(* CODESYS project T620X_PLC_CR711S_SP16p5_32bit.project
   Title: T620X PLC
   Version: 1.0.3.0
   Company: Mtech

Project tree, tasks and I/O mapping:
  SafetyPLC : CR711S SIL2, ifm electronic, order no. CR711S, version 3.2.0.0
    application Application
      libraries: ifmR360-3, * (ifm electronic); Standard, * (System); Util, * (System)
      task Task (cyclic, interval t#10ms, priority 1, watchdog t#8ms x 1) calls PLC_PRG
      global variables EVL
      program PLC_PRG [FBD]
    Communication : Communication, ifm electronic, version 3.2.0.0
      CAN : CAN, ifm electronic, version 3.2.0.0
      Ethernet : Ethernet, ifm electronic, version 3.2.0.0
    HMI : HMI, ifm electronic, version 3.2.0.0
      User_LEDs : User_LEDs, ifm electronic, version 3.2.0.0
          input  UserLED0_I AT %IB534 : LED_IEC_B_INPUT_MAPPING_TYPE  // UserLED0_I
          input  UserLED1_I : LED_IEC_B_INPUT_MAPPING_TYPE  // UserLED1_I
          input  UserLED2_I : LED_IEC_B_INPUT_MAPPING_TYPE  // UserLED2_I
          input  UserLED3_I : LED_IEC_B_INPUT_MAPPING_TYPE  // UserLED3_I
          output UserLED0_Q : LED_IEC_B_OUTPUT_MAPPING_TYPE  // User LED 0
          output UserLED1_Q : LED_IEC_B_OUTPUT_MAPPING_TYPE  // User LED 1
          output UserLED2_Q : LED_IEC_B_OUTPUT_MAPPING_TYPE  // User LED 2
          output UserLED3_Q : LED_IEC_B_OUTPUT_MAPPING_TYPE  // User LED 3
    Local_IO : Local_IO, ifm electronic, version 3.2.0.0
      Inputs : Inputs, ifm electronic, version 3.2.0.0
          input  IN0100_I : IN_MULTIFUNCTION_A_INPUT_MAPPING_TYPE  // IN0100_I
          input  IN0101_I : IN_MULTIFUNCTION_A_INPUT_MAPPING_TYPE  // IN0101_I
          input  IN0102_I : IN_MULTIFUNCTION_A_INPUT_MAPPING_TYPE  // IN0102_I
          input  IN0103_I : IN_MULTIFUNCTION_A_INPUT_MAPPING_TYPE  // IN0103_I
          input  IN0200_I : IN_MULTIFUNCTION_A_INPUT_MAPPING_TYPE  // IN0200_I
          input  IN0201_I : IN_MULTIFUNCTION_A_INPUT_MAPPING_TYPE  // IN0201_I
          input  IN0202_I : IN_MULTIFUNCTION_A_INPUT_MAPPING_TYPE  // IN0202_I
          input  IN0203_I : IN_MULTIFUNCTION_A_INPUT_MAPPING_TYPE  // IN0203_I
          input  IN0600_I : IN_MULTIFUNCTION_A_INPUT_MAPPING_TYPE  // IN0600_I
          input  IN0601_I : IN_MULTIFUNCTION_A_INPUT_MAPPING_TYPE  // IN0601_I
          input  IN0602_I : IN_MULTIFUNCTION_A_INPUT_MAPPING_TYPE  // IN0602_I
          input  IN0603_I : IN_MULTIFUNCTION_A_INPUT_MAPPING_TYPE  // IN0603_I
          input  IN0700_I : IN_MULTIFUNCTION_A_INPUT_MAPPING_TYPE  // IN0700_I
          input  IN0701_I : IN_MULTIFUNCTION_A_INPUT_MAPPING_TYPE  // IN0701_I
          input  IN0702_I : IN_MULTIFUNCTION_A_INPUT_MAPPING_TYPE  // IN0702_I
          input  IN0703_I : IN_MULTIFUNCTION_A_INPUT_MAPPING_TYPE  // IN0703_I
          input  IN0400_I : IN_RESISTOR_A_INPUT_MAPPING_TYPE  // IN0400_I
          input  IN0401_I : IN_RESISTOR_A_INPUT_MAPPING_TYPE  // IN0401_I
          input  IN0900_I : IN_RESISTOR_A_INPUT_MAPPING_TYPE  // IN0900_I
          input  IN0901_I : IN_RESISTOR_A_INPUT_MAPPING_TYPE  // IN0901_I
          input  IN0300_I : IN_DIGITAL_B_INPUT_MAPPING_TYPE  // IN0300_I
          input  IN0301_I : IN_DIGITAL_B_INPUT_MAPPING_TYPE  // IN0301_I
          input  IN0800_I : IN_DIGITAL_B_INPUT_MAPPING_TYPE  // IN0800_I
          input  IN0801_I : IN_DIGITAL_B_INPUT_MAPPING_TYPE  // IN0801_I
          input  COM_RESET_I : IN_COMMUNICATION_RESET_INPUT_MAPPING_TYPE  // COM_RESET_I
          input  IN0000_I : IN_FREQUENCY_B_CHANNEL_A_INPUT_MAPPING_TYPE  // IN0000_I
          input  IN0002_I : IN_FREQUENCY_B_CHANNEL_A_INPUT_MAPPING_TYPE  // IN0002_I
          input  IN0500_I : IN_FREQUENCY_B_CHANNEL_A_INPUT_MAPPING_TYPE  // IN0500_I
          input  IN0502_I : IN_FREQUENCY_B_CHANNEL_A_INPUT_MAPPING_TYPE  // IN0502_I
          input  IN0001_I : IN_FREQUENCY_B_CHANNEL_B_INPUT_MAPPING_TYPE  // IN0001_I
          input  IN0003_I : IN_FREQUENCY_B_CHANNEL_B_INPUT_MAPPING_TYPE  // IN0003_I
          input  IN0501_I : IN_FREQUENCY_B_CHANNEL_B_INPUT_MAPPING_TYPE  // IN0501_I
          input  IN0503_I : IN_FREQUENCY_B_CHANNEL_B_INPUT_MAPPING_TYPE  // IN0503_I
      Outputs : Outputs, ifm electronic, version 3.2.0.0
          input  OUT0006_I : OUT_PWM_40_BRIDGE_A_INPUT_MAPPING_TYPE  // OUT0006_I
          input  OUT0106_I : OUT_PWM_40_BRIDGE_A_INPUT_MAPPING_TYPE  // OUT0106_I
          input  OUT0206_I : OUT_PWM_40_BRIDGE_A_INPUT_MAPPING_TYPE  // OUT0206_I
          input  OUT0008_I : OUT_PWM_40_A_INPUT_MAPPING_TYPE  // OUT0008_I
          input  OUT0108_I : OUT_PWM_40_A_INPUT_MAPPING_TYPE  // OUT0108_I
          input  OUT0208_I : OUT_PWM_40_A_INPUT_MAPPING_TYPE  // OUT0208_I
          input  OUT0000_I : OUT_PWM_25_A_INPUT_MAPPING_TYPE  // OUT0000_I
          input  OUT0002_I : OUT_PWM_25_A_INPUT_MAPPING_TYPE  // OUT0002_I
          input  OUT0004_I : OUT_PWM_25_A_INPUT_MAPPING_TYPE  // OUT0004_I
          input  OUT0100_I : OUT_PWM_25_A_INPUT_MAPPING_TYPE  // OUT0100_I
          input  OUT0102_I : OUT_PWM_25_A_INPUT_MAPPING_TYPE  // OUT0102_I
          input  OUT0104_I : OUT_PWM_25_A_INPUT_MAPPING_TYPE  // OUT0104_I
          input  OUT0200_I : OUT_PWM_25_A_INPUT_MAPPING_TYPE  // OUT0200_I
          input  OUT0202_I : OUT_PWM_25_A_INPUT_MAPPING_TYPE  // OUT0202_I
          input  OUT0204_I : OUT_PWM_25_A_INPUT_MAPPING_TYPE  // OUT0204_I
          input  OUT3001_I : OUT_VOLTAGE_A_INPUT_MAPPING_TYPE  // OUT3001_I
          input  OUT3000_I : OUT_SUPPLY_A_INPUT_MAPPING_TYPE  // OUT3000_I
          input  OUT0001_I : OUT_PWM_25_B_INPUT_MAPPING_TYPE  // OUT0001_I
          input  OUT0003_I : OUT_PWM_25_B_INPUT_MAPPING_TYPE  // OUT0003_I
          input  OUT0005_I : OUT_PWM_25_B_INPUT_MAPPING_TYPE  // OUT0005_I
          input  OUT0101_I : OUT_PWM_25_B_INPUT_MAPPING_TYPE  // OUT0101_I
          input  OUT0103_I : OUT_PWM_25_B_INPUT_MAPPING_TYPE  // OUT0103_I
          input  OUT0105_I : OUT_PWM_25_B_INPUT_MAPPING_TYPE  // OUT0105_I
          input  OUT0201_I : OUT_PWM_25_B_INPUT_MAPPING_TYPE  // OUT0201_I
          input  OUT0203_I : OUT_PWM_25_B_INPUT_MAPPING_TYPE  // OUT0203_I
          input  OUT0205_I : OUT_PWM_25_B_INPUT_MAPPING_TYPE  // OUT0205_I
          input  OUT0007_I : OUT_PWM_40_BRIDGE_A_INPUT_MAPPING_TYPE  // OUT0007_I
          input  OUT0107_I : OUT_PWM_40_BRIDGE_A_INPUT_MAPPING_TYPE  // OUT0107_I
          input  OUT0207_I : OUT_PWM_40_BRIDGE_A_INPUT_MAPPING_TYPE  // OUT0207_I
          output OUT0006_Q : OUT_PWM_40_BRIDGE_A_OUTPUT_MAPPING_TYPE  // OUT0006_Q
          output OUT0106_Q : OUT_PWM_40_BRIDGE_A_OUTPUT_MAPPING_TYPE  // OUT0106_Q
          output OUT0206_Q : OUT_PWM_40_BRIDGE_A_OUTPUT_MAPPING_TYPE  // OUT0206_Q
          output OUT0008_Q : OUT_PWM_40_A_OUTPUT_MAPPING_TYPE  // OUT0008_Q
          output OUT0108_Q : OUT_PWM_40_A_OUTPUT_MAPPING_TYPE  // OUT0108_Q
          output OUT0208_Q : OUT_PWM_40_A_OUTPUT_MAPPING_TYPE  // OUT0208_Q
          output OUT0000_Q : OUT_PWM_25_A_OUTPUT_MAPPING_TYPE  // OUT0000_Q
          output OUT0002_Q : OUT_PWM_25_A_OUTPUT_MAPPING_TYPE  // OUT0002_Q
          output OUT0004_Q : OUT_PWM_25_A_OUTPUT_MAPPING_TYPE  // OUT0004_Q
          output OUT0100_Q : OUT_PWM_25_A_OUTPUT_MAPPING_TYPE  // OUT0100_Q
          output OUT0102_Q : OUT_PWM_25_A_OUTPUT_MAPPING_TYPE  // OUT0102_Q
          output OUT0104_Q : OUT_PWM_25_A_OUTPUT_MAPPING_TYPE  // OUT0104_Q
          output OUT0200_Q : OUT_PWM_25_A_OUTPUT_MAPPING_TYPE  // OUT0200_Q
          output OUT0202_Q : OUT_PWM_25_A_OUTPUT_MAPPING_TYPE  // OUT0202_Q
          output OUT0204_Q : OUT_PWM_25_A_OUTPUT_MAPPING_TYPE  // OUT0204_Q
          output OUT3001_Q : OUT_VOLTAGE_A_OUTPUT_MAPPING_TYPE  // OUT3001_Q
          output OUT3000_Q : OUT_SUPPLY_A_OUTPUT_MAPPING_TYPE  // OUT3000_Q
          output OUT0001_Q : OUT_PWM_25_B_OUTPUT_MAPPING_TYPE  // OUT0001_Q
          output OUT0003_Q : OUT_PWM_25_B_OUTPUT_MAPPING_TYPE  // OUT0003_Q
          output OUT0005_Q : OUT_PWM_25_B_OUTPUT_MAPPING_TYPE  // OUT0005_Q
          output OUT0101_Q : OUT_PWM_25_B_OUTPUT_MAPPING_TYPE  // OUT0101_Q
          output OUT0103_Q : OUT_PWM_25_B_OUTPUT_MAPPING_TYPE  // OUT0103_Q
          output OUT0105_Q : OUT_PWM_25_B_OUTPUT_MAPPING_TYPE  // OUT0105_Q
          output OUT0201_Q : OUT_PWM_25_B_OUTPUT_MAPPING_TYPE  // OUT0201_Q
          output OUT0203_Q : OUT_PWM_25_B_OUTPUT_MAPPING_TYPE  // OUT0203_Q
          output OUT0205_Q : OUT_PWM_25_B_OUTPUT_MAPPING_TYPE  // OUT0205_Q
          output OUT0007_Q : OUT_PWM_40_BRIDGE_A_OUTPUT_MAPPING_TYPE  // OUT0007_Q
          output OUT0107_Q : OUT_PWM_40_BRIDGE_A_OUTPUT_MAPPING_TYPE  // OUT0107_Q
          output OUT0207_Q : OUT_PWM_40_BRIDGE_A_OUTPUT_MAPPING_TYPE  // OUT0207_Q
      System_Inputs : System_Inputs, ifm electronic, version 3.2.0.0
          input  VBB30 : IN_SYSTEM_VOLTAGE_INPUT_MAPPING_TYPE  // VBB30
          input  VBB15 : IN_SYSTEM_VOLTAGE_INPUT_MAPPING_TYPE  // VBB15
          input  TemperatureBoard0 : IN_TEMPERATURE_INPUT_MAPPING_TYPE  // TemperatureBoard0
          input  TemperatureChip0 : IN_TEMPERATURE_INPUT_MAPPING_TYPE  // TemperatureChip0
      System_Outputs : System_Outputs, ifm electronic, version 3.2.0.0
          input  VBB0_SW_I : OUT_GROUP_SWITCH_INPUT_MAPPING_TYPE  // VBB0_SW_I
          input  VBB1_SW_I : OUT_GROUP_SWITCH_INPUT_MAPPING_TYPE  // VBB1_SW_I
          input  VBB2_SW_I : OUT_GROUP_SWITCH_INPUT_MAPPING_TYPE  // VBB2_SW_I
          output VBB0_SW_Q : OUT_GROUP_SWITCH_OUTPUT_MAPPING_TYPE  // VBB0_SW_Q
          output VBB1_SW_Q : OUT_GROUP_SWITCH_OUTPUT_MAPPING_TYPE  // VBB1_SW_Q
          output VBB2_SW_Q : OUT_GROUP_SWITCH_OUTPUT_MAPPING_TYPE  // VBB2_SW_Q
          output SUPPLY_SWITCH_Q : OUT_SYS_SWITCH_OUTPUT_MAPPING_TYPE  // SUPPLY_SWITCH_Q
  StandardPLC : CR711S Standard, ifm electronic, order no. CR711S, version 3.2.0.0
    application Application
      libraries: ifmR360-3, * (ifm electronic); Standard, * (System); Util, * (System); PIL Master Library, 1.0.0 (Powerhouse IRL Ltd); SLL_IFM_Version, 0.0.0.2 (SLL); SLL_IFM_CRXXXX, 0.0.0.1 (SLL); SLL Common, 0.0.0.1 (SLL); SLL_IFM_IO, 0.0.1.0 (SLL)
      task Task (cyclic, interval t#10ms, priority 1, watchdog t#8ms x 1) calls PLC_PRG_MAIN
      task Task_UDP (cyclic, interval 2 ms, priority 2, watchdog T#500MS x 1) calls UDP_MAIN
      EVC
      program PLC_Version [FBD]
      global variables NVL_UDP_TX
      Inputs/
        program Inputs [FBD]
      program UDP_MAIN [FBD]
      declarations NVL_UDP_RX
      Outputs/
        program Outputs [FBD]
        function block CRXXXX_OUTPUT_PWM_FB [FBD]: Process
      Visualisations/
        visualisation Input_IFM_PLC_CRXXXX
        visualisation Output_IFM_PLC_CRXXXX
        visualisation Output_IFM_PLC_CRXXXX_GROUP
        visualisation Inputs_Test
        visualisation Outputs_Test
      program PLC_UDP_WDT_Check [FBD]
      data type T620X_SETTINGS
      App_PLC/
        program PLC_PRG_MAIN [FBD]
        global variables GVL_APP
        Control/
          program TRACK [FBD]
          program INTERLOCKS [FBD]
        program PLC_PRG_APP [FBD]
    Communication : Communication, ifm electronic, version 3.2.0.0
      CAN : CAN, ifm electronic, version 3.2.0.0
      Ethernet : Ethernet, ifm electronic, version 3.2.0.0
    HMI : HMI, ifm electronic, version 3.2.0.0
      User_LEDs : User_LEDs, ifm electronic, version 3.2.0.0
          input  UserLED0_I : LED_IEC_B_INPUT_MAPPING_TYPE  // UserLED0_I
          input  UserLED1_I : LED_IEC_B_INPUT_MAPPING_TYPE  // UserLED1_I
          input  UserLED2_I : LED_IEC_B_INPUT_MAPPING_TYPE  // UserLED2_I
          input  UserLED3_I : LED_IEC_B_INPUT_MAPPING_TYPE  // UserLED3_I
          output UserLED0_Q : LED_IEC_B_OUTPUT_MAPPING_TYPE  // User LED 0
          output UserLED1_Q : LED_IEC_B_OUTPUT_MAPPING_TYPE  // User LED 1
          output UserLED2_Q : LED_IEC_B_OUTPUT_MAPPING_TYPE  // User LED 2
          output UserLED3_Q : LED_IEC_B_OUTPUT_MAPPING_TYPE  // User LED 3
    Local_IO : Local_IO, ifm electronic, version 3.2.0.0
      Inputs : Inputs, ifm electronic, version 3.2.0.0
          input  IN0100_I : IN_MULTIFUNCTION_A_INPUT_MAPPING_TYPE  // IN0100_I
          input  IN0101_I : IN_MULTIFUNCTION_A_INPUT_MAPPING_TYPE  // IN0101_I
          input  IN0102_I : IN_MULTIFUNCTION_A_INPUT_MAPPING_TYPE  // IN0102_I
          input  IN0103_I : IN_MULTIFUNCTION_A_INPUT_MAPPING_TYPE  // IN0103_I
          input  IN0200_I : IN_MULTIFUNCTION_A_INPUT_MAPPING_TYPE  // IN0200_I
          input  IN0201_I : IN_MULTIFUNCTION_A_INPUT_MAPPING_TYPE  // IN0201_I
          input  IN0202_I : IN_MULTIFUNCTION_A_INPUT_MAPPING_TYPE  // IN0202_I
          input  IN0203_I : IN_MULTIFUNCTION_A_INPUT_MAPPING_TYPE  // IN0203_I
          input  IN0600_I : IN_MULTIFUNCTION_A_INPUT_MAPPING_TYPE  // IN0600_I
          input  IN0601_I : IN_MULTIFUNCTION_A_INPUT_MAPPING_TYPE  // IN0601_I
          input  IN0602_I : IN_MULTIFUNCTION_A_INPUT_MAPPING_TYPE  // IN0602_I
          input  IN0603_I : IN_MULTIFUNCTION_A_INPUT_MAPPING_TYPE  // IN0603_I
          input  IN0700_I : IN_MULTIFUNCTION_A_INPUT_MAPPING_TYPE  // IN0700_I
          input  IN0701_I : IN_MULTIFUNCTION_A_INPUT_MAPPING_TYPE  // IN0701_I
          input  IN0702_I : IN_MULTIFUNCTION_A_INPUT_MAPPING_TYPE  // IN0702_I
          input  IN0703_I : IN_MULTIFUNCTION_A_INPUT_MAPPING_TYPE  // IN0703_I
          input  IN0400_I : IN_RESISTOR_A_INPUT_MAPPING_TYPE  // IN0400_I
          input  IN0401_I : IN_RESISTOR_A_INPUT_MAPPING_TYPE  // IN0401_I
          input  IN0900_I : IN_RESISTOR_A_INPUT_MAPPING_TYPE  // IN0900_I
          input  IN0901_I : IN_RESISTOR_A_INPUT_MAPPING_TYPE  // IN0901_I
          input  IN0300_I : IN_DIGITAL_B_INPUT_MAPPING_TYPE  // IN0300_I
          input  IN0301_I : IN_DIGITAL_B_INPUT_MAPPING_TYPE  // IN0301_I
          input  IN0800_I : IN_DIGITAL_B_INPUT_MAPPING_TYPE  // IN0800_I
          input  IN0801_I : IN_DIGITAL_B_INPUT_MAPPING_TYPE  // IN0801_I
          input  COM_RESET_I : IN_COMMUNICATION_RESET_INPUT_MAPPING_TYPE  // COM_RESET_I
          input  IN0000_I : IN_FREQUENCY_B_CHANNEL_A_INPUT_MAPPING_TYPE  // IN0000_I
          input  IN0002_I : IN_FREQUENCY_B_CHANNEL_A_INPUT_MAPPING_TYPE  // IN0002_I
          input  IN0500_I : IN_FREQUENCY_B_CHANNEL_A_INPUT_MAPPING_TYPE  // IN0500_I
          input  IN0502_I : IN_FREQUENCY_B_CHANNEL_A_INPUT_MAPPING_TYPE  // IN0502_I
          input  IN0001_I : IN_FREQUENCY_B_CHANNEL_B_INPUT_MAPPING_TYPE  // IN0001_I
          input  IN0003_I : IN_FREQUENCY_B_CHANNEL_B_INPUT_MAPPING_TYPE  // IN0003_I
          input  IN0501_I : IN_FREQUENCY_B_CHANNEL_B_INPUT_MAPPING_TYPE  // IN0501_I
          input  IN0503_I : IN_FREQUENCY_B_CHANNEL_B_INPUT_MAPPING_TYPE  // IN0503_I
      Outputs : Outputs, ifm electronic, version 3.2.0.0
          input  OUT0006_I : OUT_PWM_40_BRIDGE_A_INPUT_MAPPING_TYPE  // OUT0006_I
          input  OUT0106_I : OUT_PWM_40_BRIDGE_A_INPUT_MAPPING_TYPE  // OUT0106_I
          input  OUT0206_I : OUT_PWM_40_BRIDGE_A_INPUT_MAPPING_TYPE  // OUT0206_I
          input  OUT0008_I : OUT_PWM_40_A_INPUT_MAPPING_TYPE  // OUT0008_I
          input  OUT0108_I : OUT_PWM_40_A_INPUT_MAPPING_TYPE  // OUT0108_I
          input  OUT0208_I : OUT_PWM_40_A_INPUT_MAPPING_TYPE  // OUT0208_I
          input  OUT0000_I : OUT_PWM_25_A_INPUT_MAPPING_TYPE  // OUT0000_I
          input  OUT0002_I : OUT_PWM_25_A_INPUT_MAPPING_TYPE  // OUT0002_I
          input  OUT0004_I : OUT_PWM_25_A_INPUT_MAPPING_TYPE  // OUT0004_I
          input  OUT0100_I : OUT_PWM_25_A_INPUT_MAPPING_TYPE  // OUT0100_I
          input  OUT0102_I : OUT_PWM_25_A_INPUT_MAPPING_TYPE  // OUT0102_I
          input  OUT0104_I : OUT_PWM_25_A_INPUT_MAPPING_TYPE  // OUT0104_I
          input  OUT0200_I : OUT_PWM_25_A_INPUT_MAPPING_TYPE  // OUT0200_I
          input  OUT0202_I : OUT_PWM_25_A_INPUT_MAPPING_TYPE  // OUT0202_I
          input  OUT0204_I : OUT_PWM_25_A_INPUT_MAPPING_TYPE  // OUT0204_I
          input  OUT3001_I : OUT_VOLTAGE_A_INPUT_MAPPING_TYPE  // OUT3001_I
          input  OUT3000_I : OUT_SUPPLY_A_INPUT_MAPPING_TYPE  // OUT3000_I
          input  OUT0001_I : OUT_PWM_25_B_INPUT_MAPPING_TYPE  // OUT0001_I
          input  OUT0003_I : OUT_PWM_25_B_INPUT_MAPPING_TYPE  // OUT0003_I
          input  OUT0005_I : OUT_PWM_25_B_INPUT_MAPPING_TYPE  // OUT0005_I
          input  OUT0101_I : OUT_PWM_25_B_INPUT_MAPPING_TYPE  // OUT0101_I
          input  OUT0103_I : OUT_PWM_25_B_INPUT_MAPPING_TYPE  // OUT0103_I
          input  OUT0105_I : OUT_PWM_25_B_INPUT_MAPPING_TYPE  // OUT0105_I
          input  OUT0201_I : OUT_PWM_25_B_INPUT_MAPPING_TYPE  // OUT0201_I
          input  OUT0203_I : OUT_PWM_25_B_INPUT_MAPPING_TYPE  // OUT0203_I
          input  OUT0205_I : OUT_PWM_25_B_INPUT_MAPPING_TYPE  // OUT0205_I
          input  OUT0007_I : OUT_PWM_40_BRIDGE_A_INPUT_MAPPING_TYPE  // OUT0007_I
          input  OUT0107_I : OUT_PWM_40_BRIDGE_A_INPUT_MAPPING_TYPE  // OUT0107_I
          input  OUT0207_I : OUT_PWM_40_BRIDGE_A_INPUT_MAPPING_TYPE  // OUT0207_I
          output OUT0006_Q : OUT_PWM_40_BRIDGE_A_OUTPUT_MAPPING_TYPE  // OUT0006_Q
          output OUT0106_Q : OUT_PWM_40_BRIDGE_A_OUTPUT_MAPPING_TYPE  // OUT0106_Q
          output OUT0206_Q : OUT_PWM_40_BRIDGE_A_OUTPUT_MAPPING_TYPE  // OUT0206_Q
          output OUT0008_Q : OUT_PWM_40_A_OUTPUT_MAPPING_TYPE  // OUT0008_Q
          output OUT0108_Q : OUT_PWM_40_A_OUTPUT_MAPPING_TYPE  // OUT0108_Q
          output OUT0208_Q : OUT_PWM_40_A_OUTPUT_MAPPING_TYPE  // OUT0208_Q
          output OUT0000_Q : OUT_PWM_25_A_OUTPUT_MAPPING_TYPE  // OUT0000_Q
          output OUT0002_Q : OUT_PWM_25_A_OUTPUT_MAPPING_TYPE  // OUT0002_Q
          output OUT0004_Q : OUT_PWM_25_A_OUTPUT_MAPPING_TYPE  // OUT0004_Q
          output OUT0100_Q : OUT_PWM_25_A_OUTPUT_MAPPING_TYPE  // OUT0100_Q
          output OUT0102_Q : OUT_PWM_25_A_OUTPUT_MAPPING_TYPE  // OUT0102_Q
          output OUT0104_Q : OUT_PWM_25_A_OUTPUT_MAPPING_TYPE  // OUT0104_Q
          output OUT0200_Q : OUT_PWM_25_A_OUTPUT_MAPPING_TYPE  // OUT0200_Q
          output OUT0202_Q : OUT_PWM_25_A_OUTPUT_MAPPING_TYPE  // OUT0202_Q
          output OUT0204_Q : OUT_PWM_25_A_OUTPUT_MAPPING_TYPE  // OUT0204_Q
          output OUT3001_Q : OUT_VOLTAGE_A_OUTPUT_MAPPING_TYPE  // OUT3001_Q
          output OUT3000_Q : OUT_SUPPLY_A_OUTPUT_MAPPING_TYPE  // OUT3000_Q
          output OUT0001_Q : OUT_PWM_25_B_OUTPUT_MAPPING_TYPE  // OUT0001_Q
          output OUT0003_Q : OUT_PWM_25_B_OUTPUT_MAPPING_TYPE  // OUT0003_Q
          output OUT0005_Q : OUT_PWM_25_B_OUTPUT_MAPPING_TYPE  // OUT0005_Q
          output OUT0101_Q : OUT_PWM_25_B_OUTPUT_MAPPING_TYPE  // OUT0101_Q
          output OUT0103_Q : OUT_PWM_25_B_OUTPUT_MAPPING_TYPE  // OUT0103_Q
          output OUT0105_Q : OUT_PWM_25_B_OUTPUT_MAPPING_TYPE  // OUT0105_Q
          output OUT0201_Q : OUT_PWM_25_B_OUTPUT_MAPPING_TYPE  // OUT0201_Q
          output OUT0203_Q : OUT_PWM_25_B_OUTPUT_MAPPING_TYPE  // OUT0203_Q
          output OUT0205_Q : OUT_PWM_25_B_OUTPUT_MAPPING_TYPE  // OUT0205_Q
          output OUT0007_Q : OUT_PWM_40_BRIDGE_A_OUTPUT_MAPPING_TYPE  // OUT0007_Q
          output OUT0107_Q : OUT_PWM_40_BRIDGE_A_OUTPUT_MAPPING_TYPE  // OUT0107_Q
          output OUT0207_Q : OUT_PWM_40_BRIDGE_A_OUTPUT_MAPPING_TYPE  // OUT0207_Q
      System_Inputs : System_Inputs, ifm electronic, version 3.2.0.0
          input  VBB30 AT %IW251 : IN_SYSTEM_VOLTAGE_INPUT_MAPPING_TYPE  // VBB30
          input  VBB15 : IN_SYSTEM_VOLTAGE_INPUT_MAPPING_TYPE  // VBB15
          input  TemperatureBoard0 : IN_TEMPERATURE_INPUT_MAPPING_TYPE  // TemperatureBoard0
          input  TemperatureChip0 : IN_TEMPERATURE_INPUT_MAPPING_TYPE  // TemperatureChip0
      System_Outputs : System_Outputs, ifm electronic, version 3.2.0.0
          input  VBB0_SW_I : OUT_GROUP_SWITCH_INPUT_MAPPING_TYPE  // VBB0_SW_I
          input  VBB1_SW_I : OUT_GROUP_SWITCH_INPUT_MAPPING_TYPE  // VBB1_SW_I
          input  VBB2_SW_I : OUT_GROUP_SWITCH_INPUT_MAPPING_TYPE  // VBB2_SW_I
          output VBB0_SW_Q : OUT_GROUP_SWITCH_OUTPUT_MAPPING_TYPE  // VBB0_SW_Q
          output VBB1_SW_Q : OUT_GROUP_SWITCH_OUTPUT_MAPPING_TYPE  // VBB1_SW_Q
          output VBB2_SW_Q : OUT_GROUP_SWITCH_OUTPUT_MAPPING_TYPE  // VBB2_SW_Q
          output SUPPLY_SWITCH_Q : OUT_SYS_SWITCH_OUTPUT_MAPPING_TYPE  // SUPPLY_SWITCH_Q
  CR711S : CR711S, ifm electronic, order no. CR711S, version 3.2.0.0
  Project Information/
    function GetCompany [ST]
    function GetTitle [ST]
    function GetVersion [ST]
    function GetTextProperty [ST]
    function GetTextProperty2 [ST]
    function GetNumberProperty [ST]
    function GetBooleanProperty [ST]
    function GetVersionProperty [ST]
  text list GlobalTextList
*)

// StandardPLC/Application/T620X_SETTINGS
TYPE T620X_SETTINGS :
STRUCT
	FwdTime_sec: WORD;
	RevTime_sec: WORD;
	TailConvSpd_Percent: BYTE:=100;
	SideConvSpd_Percent: BYTE:=100;
	SideTransferConvSpd_Percent: BYTE:=100;
	CollectConvSpd_Percent: BYTE:=100;
	DrumSpd_Percent: BYTE:=100;
	FeederSpd_Percent: BYTE:=100;
	TailConvSpd_Min_mA: INT:=500;
	TailConvSpd_Max_mA: INT:=1450;
	SideConvSpd_Min_mA: INT:=500;
	SideConvSpd_Max_mA: INT:=1450;
	SideTransferConvSpd_Min_mA: INT:=500;
	SideTransferConvSpd_Max_mA: INT:=1450;
	CollectConvSpd_Min_mA: INT:=500;
	CollectConvSpd_Max_mA: INT:=1450;
	DrumSpd_Min_mA: INT:=500;
	DrumSpd_Max_mA: INT:=1450;
	FeederSpd_Min_mA: INT:=500;
	FeederSpd_Max_mA: INT:=1450;
	EnableDrumPressCutOut: BOOL:=TRUE;
	DrumPressReset_SP_bar: BYTE:=150;
	DrumPressHi_SP_bar: BYTE:=160;
	DrumPressHiHi_SP_bar: BYTE:=165;	
END_STRUCT
END_TYPE

// SafetyPLC/Application/EVL
(* THIS EVL IS AUTOGENERATED. DO NOT MODIFY THESE ATTRIBUTES. *)
{attribute 'location' := '16#800' }
{attribute 'linkalways'}
{attribute 'qualified_only'}
VAR_GLOBAL

END_VAR

// StandardPLC/Application/App_PLC/GVL_APP
{attribute 'qualified_only'}
VAR_GLOBAL
	Reset: BOOL;
	LED0:BYTE;
	LED1:BYTE;
	LED2:BYTE;
	LED3:BYTE;	
END_VAR

// StandardPLC/Application/NVL_UDP_TX
{attribute 'qualified_only'}
VAR_GLOBAL
	Version: SLL_IFM_Version.PLC_Version;
	System: SLL_IFM_CRXXXX.IFM_CRXXXX_System_STRUCT;
	All_Inputs: SLL_IFM_IO.CR0709_ALL_INPUTS_DATA;
	All_Outputs_Diag: SLL_IFM_IO.CR0709_ALL_OUTPUTS_DATA;	
	UDP_HB_RX_STATS: UDP_RX_STATS_HB_STRUCT;	
END_VAR

// StandardPLC/Application/NVL_UDP_RX
//This gobal variable list is received via the network.
//Sender: Imported from file '..\GVLS\NVL_UDP_HMI_TO_CR711S.gvl'
//Protocol: UDP

{attribute 'qualified_only'}
VAR_GLOBAL
	Header: IFM_HMI_Version_System_Header;
	All: SLL_IFM_IO.CR0709_ALL_OUTPUT_STATES;
	App_Settings: T620X_SETTINGS;
END_VAR

// SafetyPLC/Application/PLC_PRG
PROGRAM PLC_PRG
VAR
END_VAR

// NETWORK 1

END_PROGRAM

// StandardPLC/Application/App_PLC/PLC_PRG_MAIN
PROGRAM PLC_PRG_MAIN
VAR
	init: BOOL := TRUE;
END_VAR

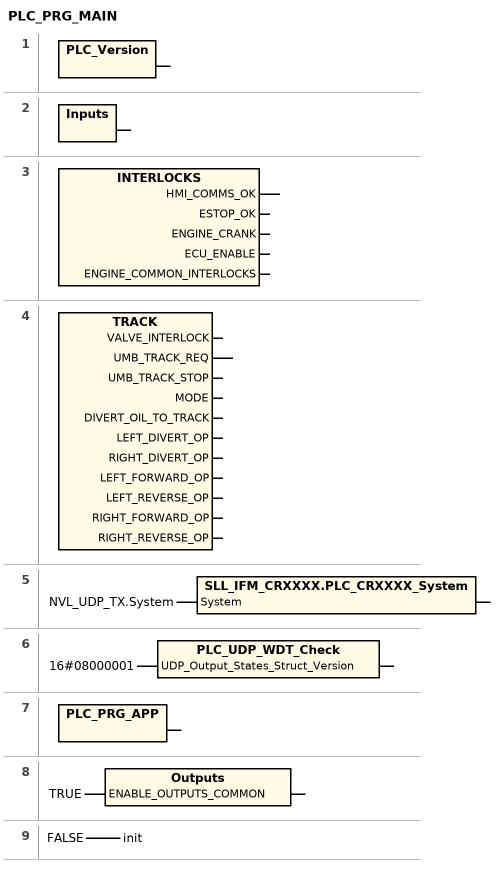
// NETWORK 1
PLC_Version();

// NETWORK 2
Inputs();

// NETWORK 3
INTERLOCKS();

// NETWORK 4
TRACK();

// NETWORK 5
SLL_IFM_CRXXXX.PLC_CRXXXX_System(System := NVL_UDP_TX.System);

// NETWORK 6
PLC_UDP_WDT_Check(UDP_Output_States_Struct_Version := 16#08000001);

// NETWORK 7
PLC_PRG_APP();

// NETWORK 8
Outputs(ENABLE_OUTPUTS_COMMON := TRUE);

// NETWORK 9
init := FALSE;

END_PROGRAM

// StandardPLC/Application/PLC_Version
PROGRAM PLC_Version
VAR
	INIT: BOOL:=TRUE;
	Tx3000: ifmrcan.CAN_Tx;	
	Tx3000_Ton: TON;
	Tx3000_Buffer: ARRAY[0..7] OF USINT := [1,0,3,0,0,0,0,0];	// 1.0.3.0
END_VAR

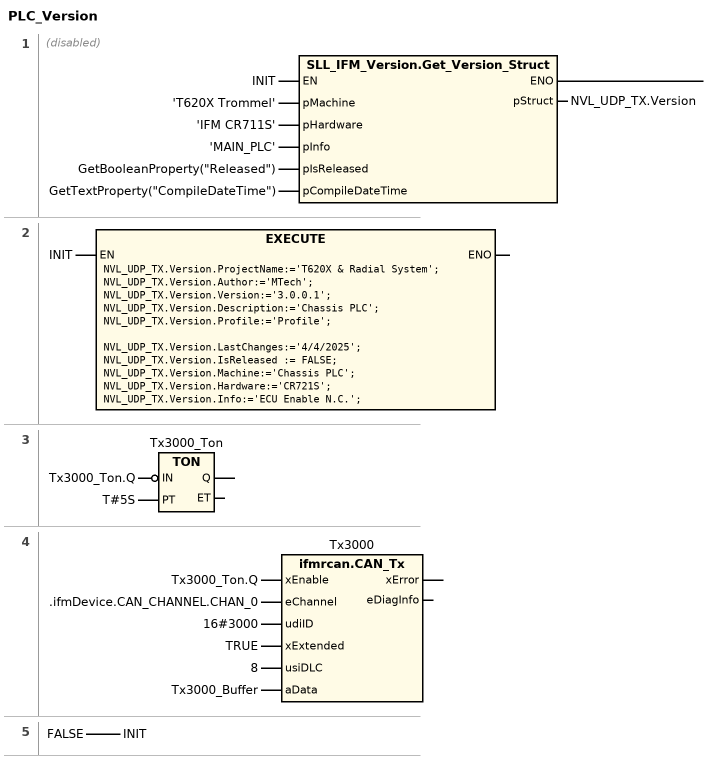
// NETWORK 1 (disabled)
// IF INIT THEN
//     SLL_IFM_Version.Get_Version_Struct(pMachine := 'T620X Trommel', pHardware := 'IFM CR711S', pInfo := 'MAIN_PLC', pIsReleased := GetBooleanProperty("Released"), pCompileDateTime := GetTextProperty("CompileDateTime"), pStruct => NVL_UDP_TX.Version);
// END_IF

// NETWORK 2
IF INIT THEN
    NVL_UDP_TX.Version.ProjectName:='T620X & Radial System';				
    NVL_UDP_TX.Version.Author:='MTech';
    NVL_UDP_TX.Version.Version:='3.0.0.1';
    NVL_UDP_TX.Version.Description:='Chassis PLC';
    NVL_UDP_TX.Version.Profile:='Profile';
    
    NVL_UDP_TX.Version.LastChanges:='4/4/2025';
    NVL_UDP_TX.Version.IsReleased := FALSE;
    NVL_UDP_TX.Version.Machine:='Chassis PLC';
    NVL_UDP_TX.Version.Hardware:='CR721S';
    NVL_UDP_TX.Version.Info:='ECU Enable N.C.';
END_IF

// NETWORK 3
Tx3000_Ton(IN := NOT Tx3000_Ton.Q, PT := T#5S); // TON

// NETWORK 4
Tx3000(
    xEnable := Tx3000_Ton.Q,
    eChannel := .ifmDevice.CAN_CHANNEL.CHAN_0,
    udiID := 16#3000,
    xExtended := TRUE,
    usiDLC := 8,
    aData := Tx3000_Buffer); // ifmrcan.CAN_Tx

// NETWORK 5
INIT := FALSE;

END_PROGRAM

// Project Information/GetBooleanProperty
// This function has been automatically generated from the project information.
{attribute 'signature_flag' := '1073741824'}
{attribute 'register_in_runtime'}
FUNCTION GetBooleanProperty : BOOL
VAR_INPUT
	stKey: WSTRING;
END_VAR

IF stKey = "Released" THEN
	GetBooleanProperty := FALSE;
ELSE
	GetBooleanProperty := FALSE;
END_IF

END_FUNCTION

// Project Information/GetTextProperty
// This function has been automatically generated from the project information.
{attribute 'signature_flag' := '1073741824'}
{attribute 'register_in_runtime'}
FUNCTION GetTextProperty : WSTRING
VAR_INPUT
	stKey: WSTRING;
END_VAR

IF stKey = "Company" THEN
	GetTextProperty := "Mtech";
ELSIF stKey = "Description" THEN
	GetTextProperty := "";
ELSIF stKey = "Project" THEN
	GetTextProperty := "T620X_PLC_CR711S_SP16p5_32bit";
ELSIF stKey = "Title" THEN
	GetTextProperty := "T620X PLC";
ELSE
	GetTextProperty := "";
END_IF

END_FUNCTION

// StandardPLC/Application/Inputs/Inputs
PROGRAM Inputs
VAR
	INPUTS_COMMON_RESET: BOOL;
	Input_FBS: SLL_IFM_IO.CR0709_ALL_INPUTS_FB;	
END_VAR

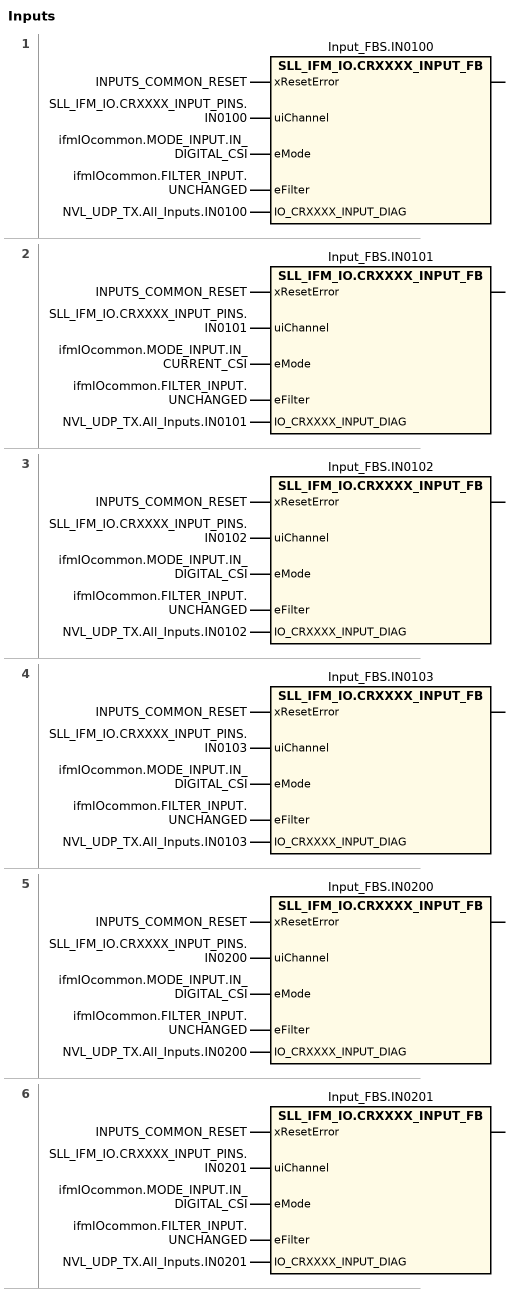
// NETWORK 1
Input_FBS.IN0100(
    xResetError := INPUTS_COMMON_RESET,
    uiChannel := SLL_IFM_IO.CRXXXX_INPUT_PINS.IN0100,
    eMode := ifmIOcommon.MODE_INPUT.IN_DIGITAL_CSI,
    eFilter := ifmIOcommon.FILTER_INPUT.UNCHANGED,
    IO_CRXXXX_INPUT_DIAG := NVL_UDP_TX.All_Inputs.IN0100); // SLL_IFM_IO.CRXXXX_INPUT_FB

// NETWORK 2
Input_FBS.IN0101(
    xResetError := INPUTS_COMMON_RESET,
    uiChannel := SLL_IFM_IO.CRXXXX_INPUT_PINS.IN0101,
    eMode := ifmIOcommon.MODE_INPUT.IN_CURRENT_CSI,
    eFilter := ifmIOcommon.FILTER_INPUT.UNCHANGED,
    IO_CRXXXX_INPUT_DIAG := NVL_UDP_TX.All_Inputs.IN0101); // SLL_IFM_IO.CRXXXX_INPUT_FB

// NETWORK 3
Input_FBS.IN0102(
    xResetError := INPUTS_COMMON_RESET,
    uiChannel := SLL_IFM_IO.CRXXXX_INPUT_PINS.IN0102,
    eMode := ifmIOcommon.MODE_INPUT.IN_DIGITAL_CSI,
    eFilter := ifmIOcommon.FILTER_INPUT.UNCHANGED,
    IO_CRXXXX_INPUT_DIAG := NVL_UDP_TX.All_Inputs.IN0102); // SLL_IFM_IO.CRXXXX_INPUT_FB

// NETWORK 4
Input_FBS.IN0103(
    xResetError := INPUTS_COMMON_RESET,
    uiChannel := SLL_IFM_IO.CRXXXX_INPUT_PINS.IN0103,
    eMode := ifmIOcommon.MODE_INPUT.IN_DIGITAL_CSI,
    eFilter := ifmIOcommon.FILTER_INPUT.UNCHANGED,
    IO_CRXXXX_INPUT_DIAG := NVL_UDP_TX.All_Inputs.IN0103); // SLL_IFM_IO.CRXXXX_INPUT_FB

// NETWORK 5
Input_FBS.IN0200(
    xResetError := INPUTS_COMMON_RESET,
    uiChannel := SLL_IFM_IO.CRXXXX_INPUT_PINS.IN0200,
    eMode := ifmIOcommon.MODE_INPUT.IN_DIGITAL_CSI,
    eFilter := ifmIOcommon.FILTER_INPUT.UNCHANGED,
    IO_CRXXXX_INPUT_DIAG := NVL_UDP_TX.All_Inputs.IN0200); // SLL_IFM_IO.CRXXXX_INPUT_FB

// NETWORK 6
Input_FBS.IN0201(
    xResetError := INPUTS_COMMON_RESET,
    uiChannel := SLL_IFM_IO.CRXXXX_INPUT_PINS.IN0201,
    eMode := ifmIOcommon.MODE_INPUT.IN_DIGITAL_CSI,
    eFilter := ifmIOcommon.FILTER_INPUT.UNCHANGED,
    IO_CRXXXX_INPUT_DIAG := NVL_UDP_TX.All_Inputs.IN0201); // SLL_IFM_IO.CRXXXX_INPUT_FB

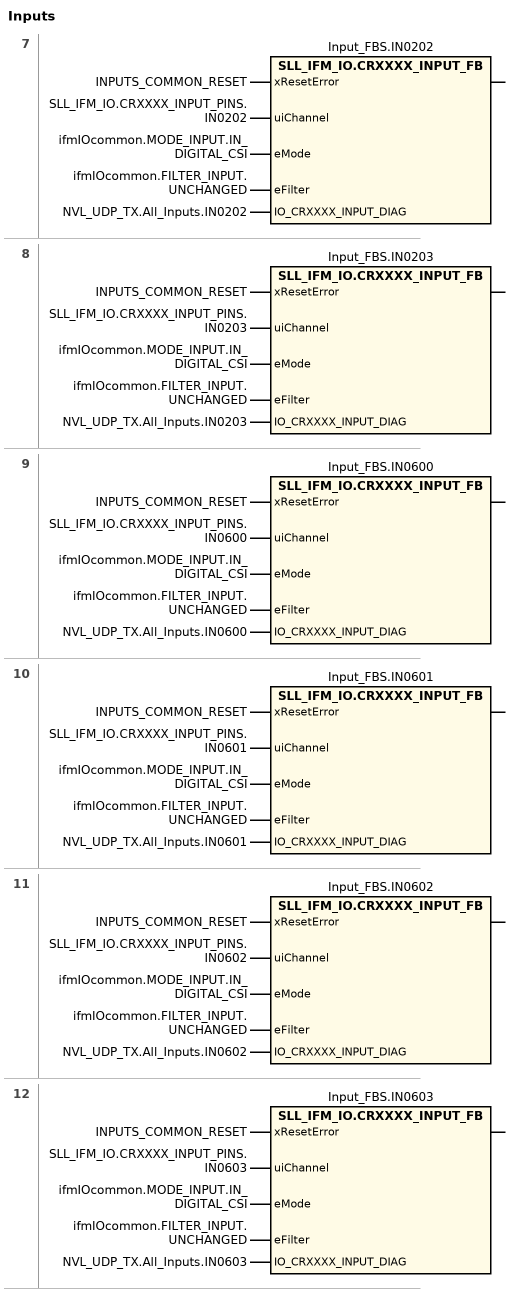
// NETWORK 7
Input_FBS.IN0202(
    xResetError := INPUTS_COMMON_RESET,
    uiChannel := SLL_IFM_IO.CRXXXX_INPUT_PINS.IN0202,
    eMode := ifmIOcommon.MODE_INPUT.IN_DIGITAL_CSI,
    eFilter := ifmIOcommon.FILTER_INPUT.UNCHANGED,
    IO_CRXXXX_INPUT_DIAG := NVL_UDP_TX.All_Inputs.IN0202); // SLL_IFM_IO.CRXXXX_INPUT_FB

// NETWORK 8
Input_FBS.IN0203(
    xResetError := INPUTS_COMMON_RESET,
    uiChannel := SLL_IFM_IO.CRXXXX_INPUT_PINS.IN0203,
    eMode := ifmIOcommon.MODE_INPUT.IN_DIGITAL_CSI,
    eFilter := ifmIOcommon.FILTER_INPUT.UNCHANGED,
    IO_CRXXXX_INPUT_DIAG := NVL_UDP_TX.All_Inputs.IN0203); // SLL_IFM_IO.CRXXXX_INPUT_FB

// NETWORK 9
Input_FBS.IN0600(
    xResetError := INPUTS_COMMON_RESET,
    uiChannel := SLL_IFM_IO.CRXXXX_INPUT_PINS.IN0600,
    eMode := ifmIOcommon.MODE_INPUT.IN_DIGITAL_CSI,
    eFilter := ifmIOcommon.FILTER_INPUT.UNCHANGED,
    IO_CRXXXX_INPUT_DIAG := NVL_UDP_TX.All_Inputs.IN0600); // SLL_IFM_IO.CRXXXX_INPUT_FB

// NETWORK 10
Input_FBS.IN0601(
    xResetError := INPUTS_COMMON_RESET,
    uiChannel := SLL_IFM_IO.CRXXXX_INPUT_PINS.IN0601,
    eMode := ifmIOcommon.MODE_INPUT.IN_DIGITAL_CSI,
    eFilter := ifmIOcommon.FILTER_INPUT.UNCHANGED,
    IO_CRXXXX_INPUT_DIAG := NVL_UDP_TX.All_Inputs.IN0601); // SLL_IFM_IO.CRXXXX_INPUT_FB

// NETWORK 11
Input_FBS.IN0602(
    xResetError := INPUTS_COMMON_RESET,
    uiChannel := SLL_IFM_IO.CRXXXX_INPUT_PINS.IN0602,
    eMode := ifmIOcommon.MODE_INPUT.IN_DIGITAL_CSI,
    eFilter := ifmIOcommon.FILTER_INPUT.UNCHANGED,
    IO_CRXXXX_INPUT_DIAG := NVL_UDP_TX.All_Inputs.IN0602); // SLL_IFM_IO.CRXXXX_INPUT_FB

// NETWORK 12
Input_FBS.IN0603(
    xResetError := INPUTS_COMMON_RESET,
    uiChannel := SLL_IFM_IO.CRXXXX_INPUT_PINS.IN0603,
    eMode := ifmIOcommon.MODE_INPUT.IN_DIGITAL_CSI,
    eFilter := ifmIOcommon.FILTER_INPUT.UNCHANGED,
    IO_CRXXXX_INPUT_DIAG := NVL_UDP_TX.All_Inputs.IN0603); // SLL_IFM_IO.CRXXXX_INPUT_FB

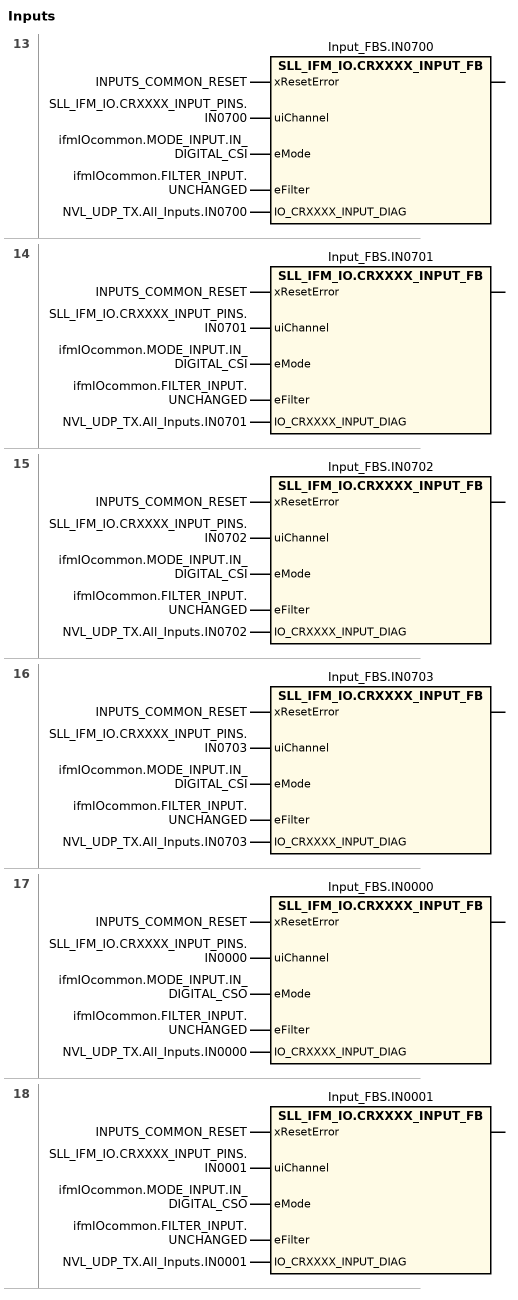
// NETWORK 13
Input_FBS.IN0700(
    xResetError := INPUTS_COMMON_RESET,
    uiChannel := SLL_IFM_IO.CRXXXX_INPUT_PINS.IN0700,
    eMode := ifmIOcommon.MODE_INPUT.IN_DIGITAL_CSI,
    eFilter := ifmIOcommon.FILTER_INPUT.UNCHANGED,
    IO_CRXXXX_INPUT_DIAG := NVL_UDP_TX.All_Inputs.IN0700); // SLL_IFM_IO.CRXXXX_INPUT_FB

// NETWORK 14
Input_FBS.IN0701(
    xResetError := INPUTS_COMMON_RESET,
    uiChannel := SLL_IFM_IO.CRXXXX_INPUT_PINS.IN0701,
    eMode := ifmIOcommon.MODE_INPUT.IN_DIGITAL_CSI,
    eFilter := ifmIOcommon.FILTER_INPUT.UNCHANGED,
    IO_CRXXXX_INPUT_DIAG := NVL_UDP_TX.All_Inputs.IN0701); // SLL_IFM_IO.CRXXXX_INPUT_FB

// NETWORK 15
Input_FBS.IN0702(
    xResetError := INPUTS_COMMON_RESET,
    uiChannel := SLL_IFM_IO.CRXXXX_INPUT_PINS.IN0702,
    eMode := ifmIOcommon.MODE_INPUT.IN_DIGITAL_CSI,
    eFilter := ifmIOcommon.FILTER_INPUT.UNCHANGED,
    IO_CRXXXX_INPUT_DIAG := NVL_UDP_TX.All_Inputs.IN0702); // SLL_IFM_IO.CRXXXX_INPUT_FB

// NETWORK 16
Input_FBS.IN0703(
    xResetError := INPUTS_COMMON_RESET,
    uiChannel := SLL_IFM_IO.CRXXXX_INPUT_PINS.IN0703,
    eMode := ifmIOcommon.MODE_INPUT.IN_DIGITAL_CSI,
    eFilter := ifmIOcommon.FILTER_INPUT.UNCHANGED,
    IO_CRXXXX_INPUT_DIAG := NVL_UDP_TX.All_Inputs.IN0703); // SLL_IFM_IO.CRXXXX_INPUT_FB

// NETWORK 17
Input_FBS.IN0000(
    xResetError := INPUTS_COMMON_RESET,
    uiChannel := SLL_IFM_IO.CRXXXX_INPUT_PINS.IN0000,
    eMode := ifmIOcommon.MODE_INPUT.IN_DIGITAL_CSO,
    eFilter := ifmIOcommon.FILTER_INPUT.UNCHANGED,
    IO_CRXXXX_INPUT_DIAG := NVL_UDP_TX.All_Inputs.IN0000); // SLL_IFM_IO.CRXXXX_INPUT_FB

// NETWORK 18
Input_FBS.IN0001(
    xResetError := INPUTS_COMMON_RESET,
    uiChannel := SLL_IFM_IO.CRXXXX_INPUT_PINS.IN0001,
    eMode := ifmIOcommon.MODE_INPUT.IN_DIGITAL_CSO,
    eFilter := ifmIOcommon.FILTER_INPUT.UNCHANGED,
    IO_CRXXXX_INPUT_DIAG := NVL_UDP_TX.All_Inputs.IN0001); // SLL_IFM_IO.CRXXXX_INPUT_FB

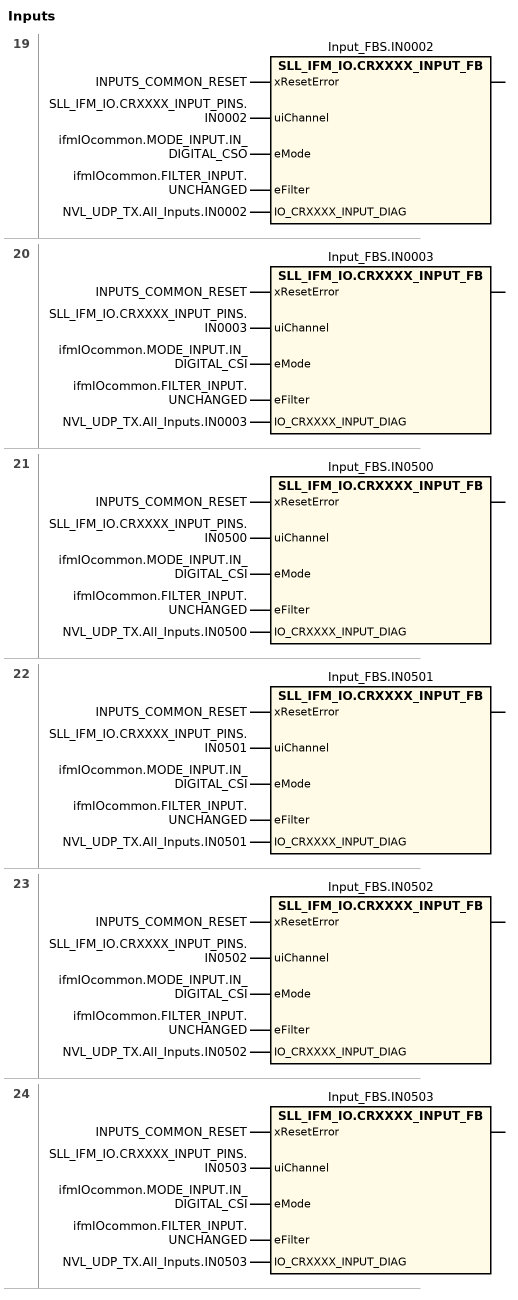
// NETWORK 19
Input_FBS.IN0002(
    xResetError := INPUTS_COMMON_RESET,
    uiChannel := SLL_IFM_IO.CRXXXX_INPUT_PINS.IN0002,
    eMode := ifmIOcommon.MODE_INPUT.IN_DIGITAL_CSO,
    eFilter := ifmIOcommon.FILTER_INPUT.UNCHANGED,
    IO_CRXXXX_INPUT_DIAG := NVL_UDP_TX.All_Inputs.IN0002); // SLL_IFM_IO.CRXXXX_INPUT_FB

// NETWORK 20
Input_FBS.IN0003(
    xResetError := INPUTS_COMMON_RESET,
    uiChannel := SLL_IFM_IO.CRXXXX_INPUT_PINS.IN0003,
    eMode := ifmIOcommon.MODE_INPUT.IN_DIGITAL_CSI,
    eFilter := ifmIOcommon.FILTER_INPUT.UNCHANGED,
    IO_CRXXXX_INPUT_DIAG := NVL_UDP_TX.All_Inputs.IN0003); // SLL_IFM_IO.CRXXXX_INPUT_FB

// NETWORK 21
Input_FBS.IN0500(
    xResetError := INPUTS_COMMON_RESET,
    uiChannel := SLL_IFM_IO.CRXXXX_INPUT_PINS.IN0500,
    eMode := ifmIOcommon.MODE_INPUT.IN_DIGITAL_CSI,
    eFilter := ifmIOcommon.FILTER_INPUT.UNCHANGED,
    IO_CRXXXX_INPUT_DIAG := NVL_UDP_TX.All_Inputs.IN0500); // SLL_IFM_IO.CRXXXX_INPUT_FB

// NETWORK 22
Input_FBS.IN0501(
    xResetError := INPUTS_COMMON_RESET,
    uiChannel := SLL_IFM_IO.CRXXXX_INPUT_PINS.IN0501,
    eMode := ifmIOcommon.MODE_INPUT.IN_DIGITAL_CSI,
    eFilter := ifmIOcommon.FILTER_INPUT.UNCHANGED,
    IO_CRXXXX_INPUT_DIAG := NVL_UDP_TX.All_Inputs.IN0501); // SLL_IFM_IO.CRXXXX_INPUT_FB

// NETWORK 23
Input_FBS.IN0502(
    xResetError := INPUTS_COMMON_RESET,
    uiChannel := SLL_IFM_IO.CRXXXX_INPUT_PINS.IN0502,
    eMode := ifmIOcommon.MODE_INPUT.IN_DIGITAL_CSI,
    eFilter := ifmIOcommon.FILTER_INPUT.UNCHANGED,
    IO_CRXXXX_INPUT_DIAG := NVL_UDP_TX.All_Inputs.IN0502); // SLL_IFM_IO.CRXXXX_INPUT_FB

// NETWORK 24
Input_FBS.IN0503(
    xResetError := INPUTS_COMMON_RESET,
    uiChannel := SLL_IFM_IO.CRXXXX_INPUT_PINS.IN0503,
    eMode := ifmIOcommon.MODE_INPUT.IN_DIGITAL_CSI,
    eFilter := ifmIOcommon.FILTER_INPUT.UNCHANGED,
    IO_CRXXXX_INPUT_DIAG := NVL_UDP_TX.All_Inputs.IN0503); // SLL_IFM_IO.CRXXXX_INPUT_FB

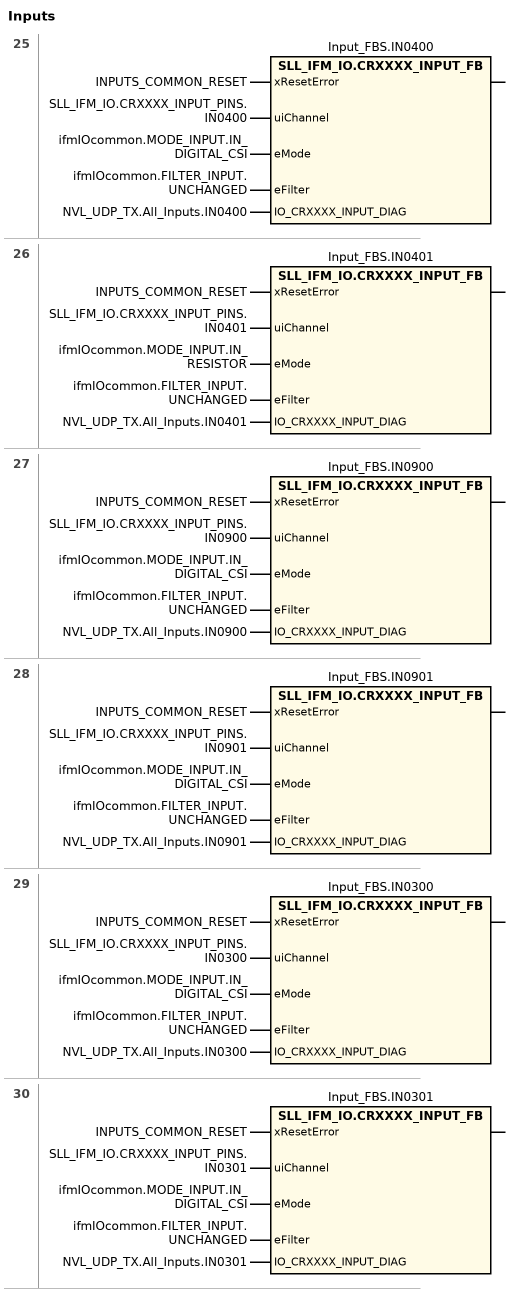
// NETWORK 25
Input_FBS.IN0400(
    xResetError := INPUTS_COMMON_RESET,
    uiChannel := SLL_IFM_IO.CRXXXX_INPUT_PINS.IN0400,
    eMode := ifmIOcommon.MODE_INPUT.IN_DIGITAL_CSI,
    eFilter := ifmIOcommon.FILTER_INPUT.UNCHANGED,
    IO_CRXXXX_INPUT_DIAG := NVL_UDP_TX.All_Inputs.IN0400); // SLL_IFM_IO.CRXXXX_INPUT_FB

// NETWORK 26
Input_FBS.IN0401(
    xResetError := INPUTS_COMMON_RESET,
    uiChannel := SLL_IFM_IO.CRXXXX_INPUT_PINS.IN0401,
    eMode := ifmIOcommon.MODE_INPUT.IN_RESISTOR,
    eFilter := ifmIOcommon.FILTER_INPUT.UNCHANGED,
    IO_CRXXXX_INPUT_DIAG := NVL_UDP_TX.All_Inputs.IN0401); // SLL_IFM_IO.CRXXXX_INPUT_FB

// NETWORK 27
Input_FBS.IN0900(
    xResetError := INPUTS_COMMON_RESET,
    uiChannel := SLL_IFM_IO.CRXXXX_INPUT_PINS.IN0900,
    eMode := ifmIOcommon.MODE_INPUT.IN_DIGITAL_CSI,
    eFilter := ifmIOcommon.FILTER_INPUT.UNCHANGED,
    IO_CRXXXX_INPUT_DIAG := NVL_UDP_TX.All_Inputs.IN0900); // SLL_IFM_IO.CRXXXX_INPUT_FB

// NETWORK 28
Input_FBS.IN0901(
    xResetError := INPUTS_COMMON_RESET,
    uiChannel := SLL_IFM_IO.CRXXXX_INPUT_PINS.IN0901,
    eMode := ifmIOcommon.MODE_INPUT.IN_DIGITAL_CSI,
    eFilter := ifmIOcommon.FILTER_INPUT.UNCHANGED,
    IO_CRXXXX_INPUT_DIAG := NVL_UDP_TX.All_Inputs.IN0901); // SLL_IFM_IO.CRXXXX_INPUT_FB

// NETWORK 29
Input_FBS.IN0300(
    xResetError := INPUTS_COMMON_RESET,
    uiChannel := SLL_IFM_IO.CRXXXX_INPUT_PINS.IN0300,
    eMode := ifmIOcommon.MODE_INPUT.IN_DIGITAL_CSI,
    eFilter := ifmIOcommon.FILTER_INPUT.UNCHANGED,
    IO_CRXXXX_INPUT_DIAG := NVL_UDP_TX.All_Inputs.IN0300); // SLL_IFM_IO.CRXXXX_INPUT_FB

// NETWORK 30
Input_FBS.IN0301(
    xResetError := INPUTS_COMMON_RESET,
    uiChannel := SLL_IFM_IO.CRXXXX_INPUT_PINS.IN0301,
    eMode := ifmIOcommon.MODE_INPUT.IN_DIGITAL_CSI,
    eFilter := ifmIOcommon.FILTER_INPUT.UNCHANGED,
    IO_CRXXXX_INPUT_DIAG := NVL_UDP_TX.All_Inputs.IN0301); // SLL_IFM_IO.CRXXXX_INPUT_FB

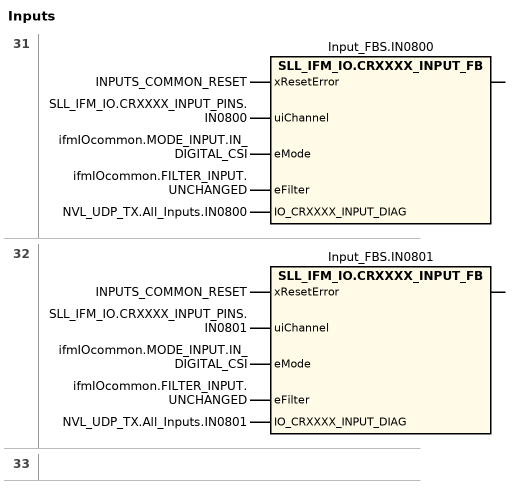
// NETWORK 31
Input_FBS.IN0800(
    xResetError := INPUTS_COMMON_RESET,
    uiChannel := SLL_IFM_IO.CRXXXX_INPUT_PINS.IN0800,
    eMode := ifmIOcommon.MODE_INPUT.IN_DIGITAL_CSI,
    eFilter := ifmIOcommon.FILTER_INPUT.UNCHANGED,
    IO_CRXXXX_INPUT_DIAG := NVL_UDP_TX.All_Inputs.IN0800); // SLL_IFM_IO.CRXXXX_INPUT_FB

// NETWORK 32
Input_FBS.IN0801(
    xResetError := INPUTS_COMMON_RESET,
    uiChannel := SLL_IFM_IO.CRXXXX_INPUT_PINS.IN0801,
    eMode := ifmIOcommon.MODE_INPUT.IN_DIGITAL_CSI,
    eFilter := ifmIOcommon.FILTER_INPUT.UNCHANGED,
    IO_CRXXXX_INPUT_DIAG := NVL_UDP_TX.All_Inputs.IN0801); // SLL_IFM_IO.CRXXXX_INPUT_FB

// NETWORK 33

END_PROGRAM

// StandardPLC/Application/App_PLC/Control/INTERLOCKS
PROGRAM INTERLOCKS
VAR
	Engine_Running_SET_TON: TON;
	ECU_ENABLE_FUNC: BOOL;
	ENGINE_CRANKING_FEEDBACK: BOOL;
	ENGINE_CRANKING_FEEDBACK_TON: TON;
	ENGINE_CRANKING_FEEDBACK_TOF: TOF;
	DUTY_CYCLE_OP_RESET:DUTY_CYCLE;
END_VAR
VAR_OUTPUT
	HMI_COMMS_OK: BOOL;
	ESTOP_OK: BOOL;
	ENGINE_CRANK: BOOL;
	ECU_ENABLE: BOOL;
	ENGINE_COMMON_INTERLOCKS: BOOL;
	OP_RESET: BOOL;
	ENGINE_RUNNING: BOOL;
END_VAR

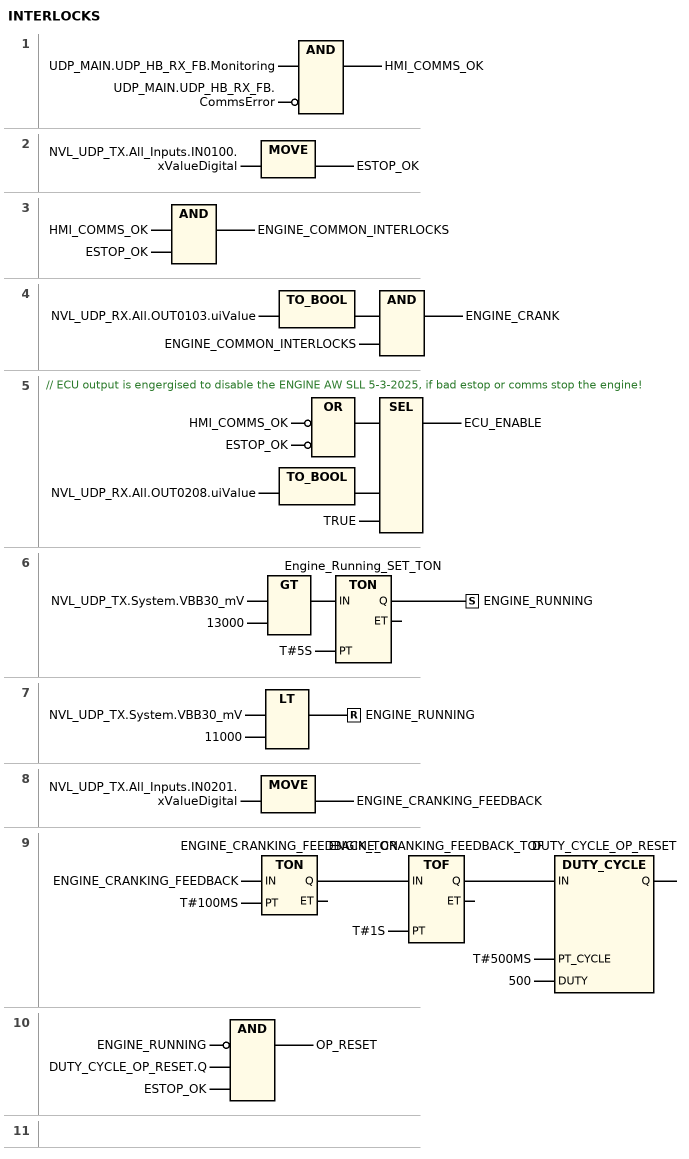
// NETWORK 1
HMI_COMMS_OK := UDP_MAIN.UDP_HB_RX_FB.Monitoring AND NOT UDP_MAIN.UDP_HB_RX_FB.CommsError;

// NETWORK 2
ESTOP_OK := NVL_UDP_TX.All_Inputs.IN0100.xValueDigital;

// NETWORK 3
ENGINE_COMMON_INTERLOCKS := HMI_COMMS_OK AND ESTOP_OK;

// NETWORK 4
ENGINE_CRANK := TO_BOOL(NVL_UDP_RX.All.OUT0103.uiValue) AND ENGINE_COMMON_INTERLOCKS;

// NETWORK 5
// // ECU output is engergised to disable the ENGINE AW SLL 5-3-2025, if bad estop or comms stop the engine!
ECU_ENABLE := SEL(NOT HMI_COMMS_OK OR NOT ESTOP_OK, TO_BOOL(NVL_UDP_RX.All.OUT0208.uiValue), TRUE);

// NETWORK 6
Engine_Running_SET_TON(IN := NVL_UDP_TX.System.VBB30_mV > 13000, PT := T#5S); // TON
ENGINE_RUNNING S= Engine_Running_SET_TON.Q;

// NETWORK 7
ENGINE_RUNNING R= NVL_UDP_TX.System.VBB30_mV < 11000;

// NETWORK 8
ENGINE_CRANKING_FEEDBACK := NVL_UDP_TX.All_Inputs.IN0201.xValueDigital;

// NETWORK 9
ENGINE_CRANKING_FEEDBACK_TON(IN := ENGINE_CRANKING_FEEDBACK, PT := T#100MS); // TON
ENGINE_CRANKING_FEEDBACK_TOF(IN := ENGINE_CRANKING_FEEDBACK_TON.Q, PT := T#1S); // TOF
DUTY_CYCLE_OP_RESET(IN := ENGINE_CRANKING_FEEDBACK_TOF.Q, PT_CYCLE := T#500MS, DUTY := 500); // DUTY_CYCLE

// NETWORK 10
OP_RESET := NOT ENGINE_RUNNING AND DUTY_CYCLE_OP_RESET.Q AND ESTOP_OK;

// NETWORK 11

END_PROGRAM

// StandardPLC/Application/UDP_MAIN
PROGRAM UDP_MAIN
VAR
	UDP_HB_RX_FB: UDP_RX_CHECK_HB_FB;
	STATS: UDP_RX_STATS_HB_STRUCT;
	
	UDP_RX_MONITORING_MS: DINT :=8000;
	UDP_RX_WARNING_DIFF_THRESHOLD: DINT := 400;
	UDP_RX_ERROR_DIFF_THRESHOLD: DINT := 500;
	UDP_RX_WARNING_FROZEN_THRESHOLD: DINT := 400;
	UDP_RX_ERROR_FROZEN_THRESHOLD: DINT :=500;
	UDP_RX_ERROR_MISSING_MS: DINT :=1000;
	UDP_RX_ERROR_RECOVERY_MS: DINT :=3000;
	
	RESET_TP: TP;
	RESET_TON: TON;	
END_VAR

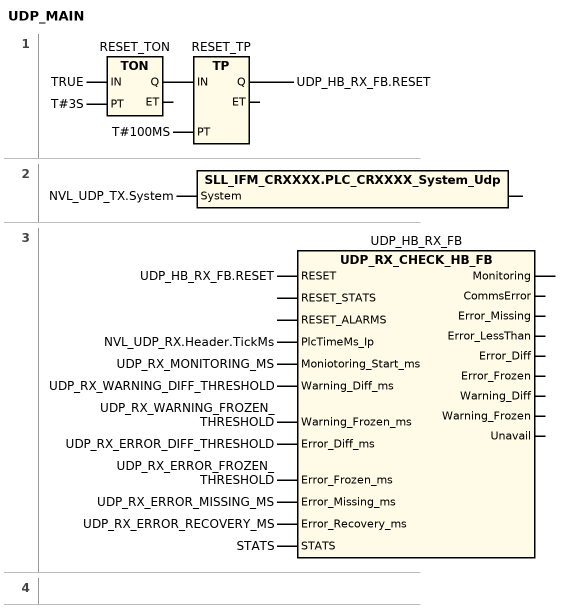
// NETWORK 1
RESET_TON(IN := TRUE, PT := T#3S); // TON
RESET_TP(IN := RESET_TON.Q, PT := T#100MS); // TP
UDP_HB_RX_FB.RESET := RESET_TP.Q;

// NETWORK 2
SLL_IFM_CRXXXX.PLC_CRXXXX_System_Udp(System := NVL_UDP_TX.System);

// NETWORK 3
UDP_HB_RX_FB(
    RESET := UDP_HB_RX_FB.RESET,
    PlcTimeMs_Ip := NVL_UDP_RX.Header.TickMs,
    Moniotoring_Start_ms := UDP_RX_MONITORING_MS,
    Warning_Diff_ms := UDP_RX_WARNING_DIFF_THRESHOLD,
    Warning_Frozen_ms := UDP_RX_WARNING_FROZEN_THRESHOLD,
    Error_Diff_ms := UDP_RX_ERROR_DIFF_THRESHOLD,
    Error_Frozen_ms := UDP_RX_ERROR_FROZEN_THRESHOLD,
    Error_Missing_ms := UDP_RX_ERROR_MISSING_MS,
    Error_Recovery_ms := UDP_RX_ERROR_RECOVERY_MS,
    STATS := STATS); // UDP_RX_CHECK_HB_FB

// NETWORK 4

END_PROGRAM

// StandardPLC/Application/App_PLC/Control/TRACK
PROGRAM TRACK
VAR
	RTF_REQ: BOOL;
	RTR_REQ: BOOL;
	LTF_REQ: BOOL;
	LTR_REQ: BOOL;	
END_VAR

VAR_OUTPUT
	VALVE_INTERLOCK: BOOL; 
	UMB_TRACK_REQ: BOOL;
	UMB_TRACK_STOP: BOOL;	
	MODE: BOOL;
	DIVERT_OIL_TO_TRACK: BOOL;
	LEFT_DIVERT_OP: BOOL;
	RIGHT_DIVERT_OP: BOOL;
	LEFT_FORWARD_OP: BOOL;
	LEFT_REVERSE_OP: BOOL;
	RIGHT_FORWARD_OP: BOOL;
	RIGHT_REVERSE_OP: BOOL;
END_VAR

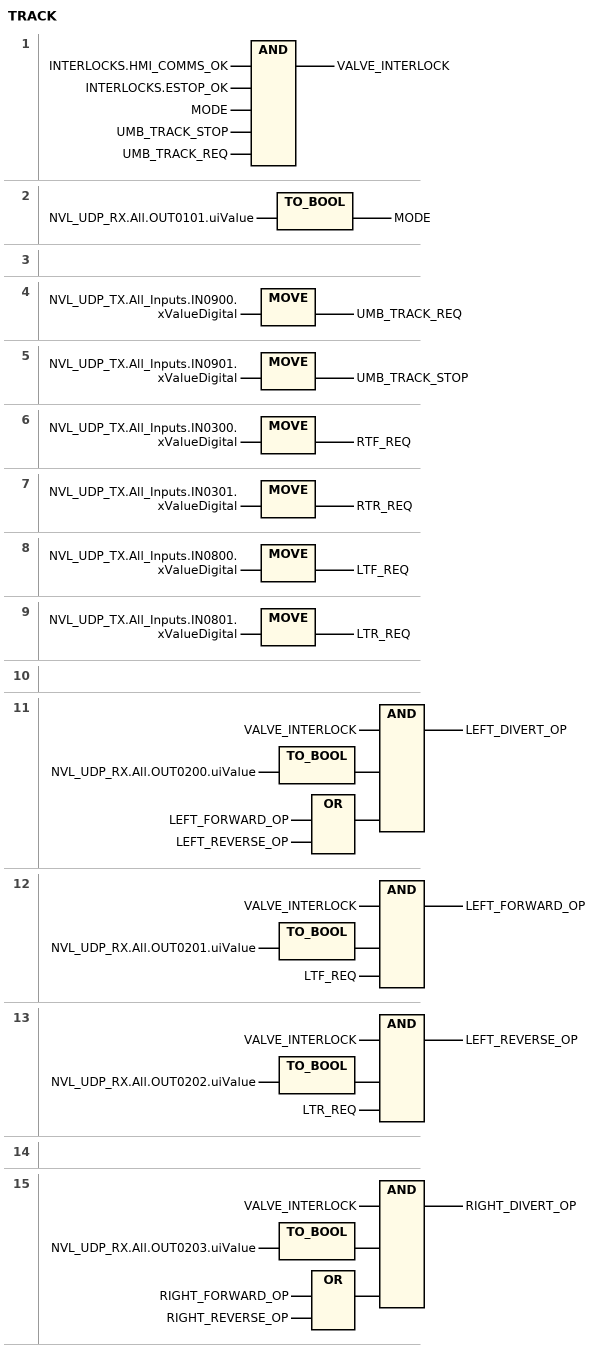
// NETWORK 1
VALVE_INTERLOCK := INTERLOCKS.HMI_COMMS_OK AND INTERLOCKS.ESTOP_OK AND MODE AND UMB_TRACK_STOP AND UMB_TRACK_REQ;

// NETWORK 2
MODE := TO_BOOL(NVL_UDP_RX.All.OUT0101.uiValue);

// NETWORK 3

// NETWORK 4
UMB_TRACK_REQ := NVL_UDP_TX.All_Inputs.IN0900.xValueDigital;

// NETWORK 5
UMB_TRACK_STOP := NVL_UDP_TX.All_Inputs.IN0901.xValueDigital;

// NETWORK 6
RTF_REQ := NVL_UDP_TX.All_Inputs.IN0300.xValueDigital;

// NETWORK 7
RTR_REQ := NVL_UDP_TX.All_Inputs.IN0301.xValueDigital;

// NETWORK 8
LTF_REQ := NVL_UDP_TX.All_Inputs.IN0800.xValueDigital;

// NETWORK 9
LTR_REQ := NVL_UDP_TX.All_Inputs.IN0801.xValueDigital;

// NETWORK 10

// NETWORK 11
LEFT_DIVERT_OP := VALVE_INTERLOCK AND TO_BOOL(NVL_UDP_RX.All.OUT0200.uiValue) AND (LEFT_FORWARD_OP OR LEFT_REVERSE_OP);

// NETWORK 12
LEFT_FORWARD_OP := VALVE_INTERLOCK AND TO_BOOL(NVL_UDP_RX.All.OUT0201.uiValue) AND LTF_REQ;

// NETWORK 13
LEFT_REVERSE_OP := VALVE_INTERLOCK AND TO_BOOL(NVL_UDP_RX.All.OUT0202.uiValue) AND LTR_REQ;

// NETWORK 14

// NETWORK 15
RIGHT_DIVERT_OP := VALVE_INTERLOCK AND TO_BOOL(NVL_UDP_RX.All.OUT0203.uiValue) AND (RIGHT_FORWARD_OP OR RIGHT_REVERSE_OP);

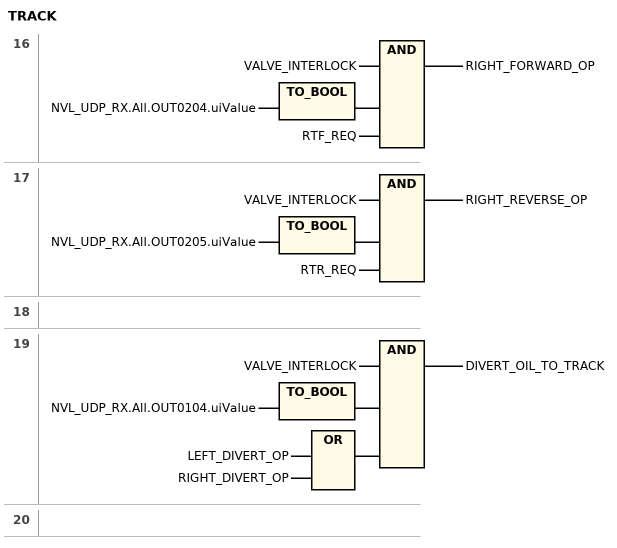
// NETWORK 16
RIGHT_FORWARD_OP := VALVE_INTERLOCK AND TO_BOOL(NVL_UDP_RX.All.OUT0204.uiValue) AND RTF_REQ;

// NETWORK 17
RIGHT_REVERSE_OP := VALVE_INTERLOCK AND TO_BOOL(NVL_UDP_RX.All.OUT0205.uiValue) AND RTR_REQ;

// NETWORK 18

// NETWORK 19
DIVERT_OIL_TO_TRACK := VALVE_INTERLOCK AND TO_BOOL(NVL_UDP_RX.All.OUT0104.uiValue) AND (LEFT_DIVERT_OP OR RIGHT_DIVERT_OP);

// NETWORK 20

END_PROGRAM

// StandardPLC/Application/PLC_UDP_WDT_Check
PROGRAM PLC_UDP_WDT_Check
VAR_INPUT
	UDP_Output_States_Struct_Version: DWORD;
END_VAR
VAR
	Local_Outputs_Test: BOOL:=0;
	Local_Outputs_Test_State: BOOL := TRUE;

	TEST_LED0_COLOUR_1: BYTE:=4;	
	TEST_LED1_COLOUR_1: BYTE:=2;
	TEST_LED2_COLOUR_1: BYTE:=1;	
END_VAR
VAR // added by the converter: edge detectors and wires of the graphical bodies
    _rt1 : R_TRIG;
END_VAR

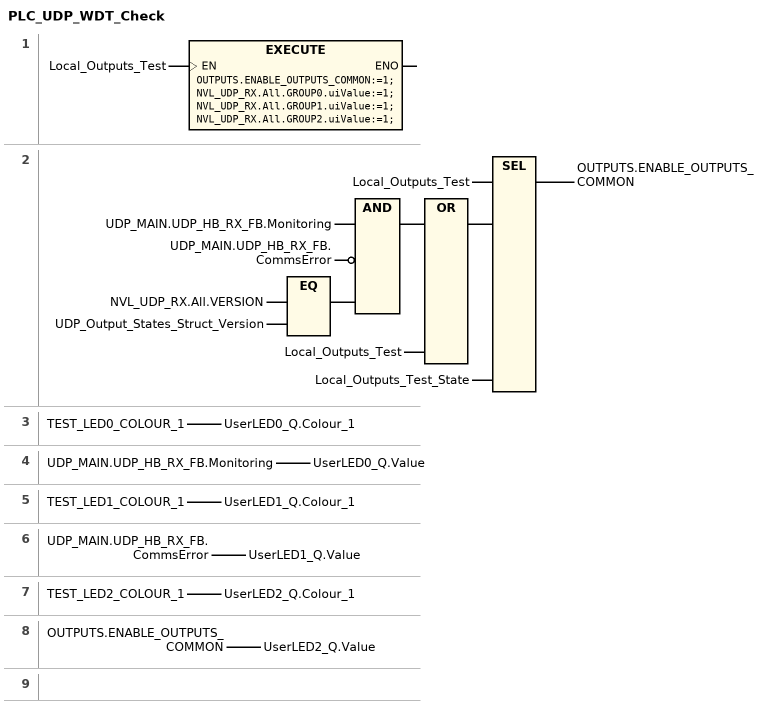
// NETWORK 1
_rt1(CLK := Local_Outputs_Test);
IF _rt1.Q THEN
    OUTPUTS.ENABLE_OUTPUTS_COMMON:=1;
    NVL_UDP_RX.All.GROUP0.uiValue:=1;
    NVL_UDP_RX.All.GROUP1.uiValue:=1;
    NVL_UDP_RX.All.GROUP2.uiValue:=1;
END_IF

// NETWORK 2
OUTPUTS.ENABLE_OUTPUTS_COMMON := SEL(Local_Outputs_Test, UDP_MAIN.UDP_HB_RX_FB.Monitoring AND NOT UDP_MAIN.UDP_HB_RX_FB.CommsError AND NVL_UDP_RX.All.VERSION = UDP_Output_States_Struct_Version OR Local_Outputs_Test, Local_Outputs_Test_State);

// NETWORK 3
UserLED0_Q.Colour_1 := TEST_LED0_COLOUR_1;

// NETWORK 4
UserLED0_Q.Value := UDP_MAIN.UDP_HB_RX_FB.Monitoring;

// NETWORK 5
UserLED1_Q.Colour_1 := TEST_LED1_COLOUR_1;

// NETWORK 6
UserLED1_Q.Value := UDP_MAIN.UDP_HB_RX_FB.CommsError;

// NETWORK 7
UserLED2_Q.Colour_1 := TEST_LED2_COLOUR_1;

// NETWORK 8
UserLED2_Q.Value := OUTPUTS.ENABLE_OUTPUTS_COMMON;

// NETWORK 9

END_PROGRAM

// StandardPLC/Application/Outputs/Outputs
PROGRAM Outputs
VAR_INPUT
	ENABLE_OUTPUTS_COMMON: BOOL;	
END_VAR
VAR
	INIT:BOOL:=TRUE;
	OUT3XXXX_GROUP_DUMMY: CRXXXX_OUTPUT_GROUP_DATA;
	
	OUTPUTS_COMMON_RESET: BOOL;
	OUTPUTS_COMMON_GROUP_OP_RESET: BOOL;
	Output_FBS: SLL_IFM_IO.CR0709_ALL_OUTPUTS_FB;
	
	OUT0000_Output: CRXXXX_OUTPUT_PWM_FB;
	OUT0002_Output: CRXXXX_OUTPUT_PWM_FB;
	OUT0004_Output: CRXXXX_OUTPUT_PWM_FB;
	OUT0007_Output: CRXXXX_OUTPUT_PWM_FB;
	OUT0100_Output: CRXXXX_OUTPUT_PWM_FB;
	OUT0102_Output: CRXXXX_OUTPUT_PWM_FB;	
		
	LOCAL_RESET:BOOL;
END_VAR

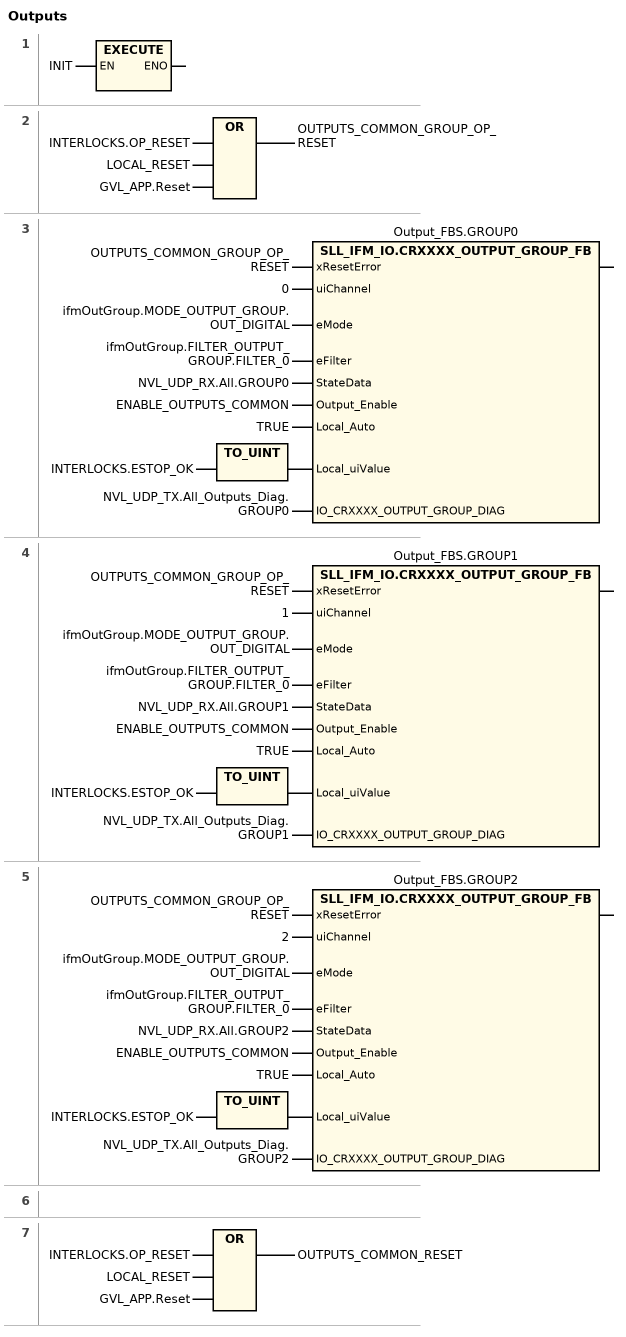
// NETWORK 1
IF INIT THEN  END_IF

// NETWORK 2
OUTPUTS_COMMON_GROUP_OP_RESET := INTERLOCKS.OP_RESET OR LOCAL_RESET OR GVL_APP.Reset;

// NETWORK 3
Output_FBS.GROUP0(
    xResetError := OUTPUTS_COMMON_GROUP_OP_RESET,
    uiChannel := 0,
    eMode := ifmOutGroup.MODE_OUTPUT_GROUP.OUT_DIGITAL,
    eFilter := ifmOutGroup.FILTER_OUTPUT_GROUP.FILTER_0,
    StateData := NVL_UDP_RX.All.GROUP0,
    Output_Enable := ENABLE_OUTPUTS_COMMON,
    Local_Auto := TRUE,
    Local_uiValue := TO_UINT(INTERLOCKS.ESTOP_OK),
    IO_CRXXXX_OUTPUT_GROUP_DIAG := NVL_UDP_TX.All_Outputs_Diag.GROUP0); // SLL_IFM_IO.CRXXXX_OUTPUT_GROUP_FB

// NETWORK 4
Output_FBS.GROUP1(
    xResetError := OUTPUTS_COMMON_GROUP_OP_RESET,
    uiChannel := 1,
    eMode := ifmOutGroup.MODE_OUTPUT_GROUP.OUT_DIGITAL,
    eFilter := ifmOutGroup.FILTER_OUTPUT_GROUP.FILTER_0,
    StateData := NVL_UDP_RX.All.GROUP1,
    Output_Enable := ENABLE_OUTPUTS_COMMON,
    Local_Auto := TRUE,
    Local_uiValue := TO_UINT(INTERLOCKS.ESTOP_OK),
    IO_CRXXXX_OUTPUT_GROUP_DIAG := NVL_UDP_TX.All_Outputs_Diag.GROUP1); // SLL_IFM_IO.CRXXXX_OUTPUT_GROUP_FB

// NETWORK 5
Output_FBS.GROUP2(
    xResetError := OUTPUTS_COMMON_GROUP_OP_RESET,
    uiChannel := 2,
    eMode := ifmOutGroup.MODE_OUTPUT_GROUP.OUT_DIGITAL,
    eFilter := ifmOutGroup.FILTER_OUTPUT_GROUP.FILTER_0,
    StateData := NVL_UDP_RX.All.GROUP2,
    Output_Enable := ENABLE_OUTPUTS_COMMON,
    Local_Auto := TRUE,
    Local_uiValue := TO_UINT(INTERLOCKS.ESTOP_OK),
    IO_CRXXXX_OUTPUT_GROUP_DIAG := NVL_UDP_TX.All_Outputs_Diag.GROUP2); // SLL_IFM_IO.CRXXXX_OUTPUT_GROUP_FB

// NETWORK 6

// NETWORK 7
OUTPUTS_COMMON_RESET := INTERLOCKS.OP_RESET OR LOCAL_RESET OR GVL_APP.Reset;

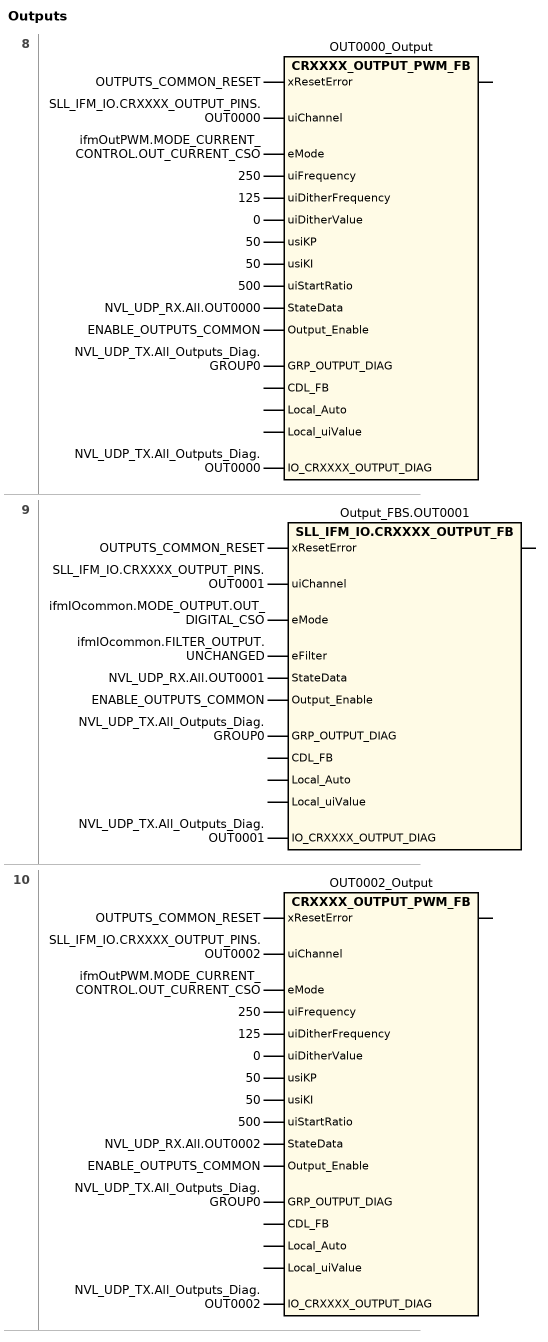
// NETWORK 8
OUT0000_Output(
    xResetError := OUTPUTS_COMMON_RESET,
    uiChannel := SLL_IFM_IO.CRXXXX_OUTPUT_PINS.OUT0000,
    eMode := ifmOutPWM.MODE_CURRENT_CONTROL.OUT_CURRENT_CSO,
    uiFrequency := 250,
    uiDitherFrequency := 125,
    uiDitherValue := 0,
    usiKP := 50,
    usiKI := 50,
    uiStartRatio := 500,
    StateData := NVL_UDP_RX.All.OUT0000,
    Output_Enable := ENABLE_OUTPUTS_COMMON,
    GRP_OUTPUT_DIAG := NVL_UDP_TX.All_Outputs_Diag.GROUP0,
    IO_CRXXXX_OUTPUT_DIAG := NVL_UDP_TX.All_Outputs_Diag.OUT0000); // CRXXXX_OUTPUT_PWM_FB

// NETWORK 9
Output_FBS.OUT0001(
    xResetError := OUTPUTS_COMMON_RESET,
    uiChannel := SLL_IFM_IO.CRXXXX_OUTPUT_PINS.OUT0001,
    eMode := ifmIOcommon.MODE_OUTPUT.OUT_DIGITAL_CSO,
    eFilter := ifmIOcommon.FILTER_OUTPUT.UNCHANGED,
    StateData := NVL_UDP_RX.All.OUT0001,
    Output_Enable := ENABLE_OUTPUTS_COMMON,
    GRP_OUTPUT_DIAG := NVL_UDP_TX.All_Outputs_Diag.GROUP0,
    IO_CRXXXX_OUTPUT_DIAG := NVL_UDP_TX.All_Outputs_Diag.OUT0001); // SLL_IFM_IO.CRXXXX_OUTPUT_FB

// NETWORK 10
OUT0002_Output(
    xResetError := OUTPUTS_COMMON_RESET,
    uiChannel := SLL_IFM_IO.CRXXXX_OUTPUT_PINS.OUT0002,
    eMode := ifmOutPWM.MODE_CURRENT_CONTROL.OUT_CURRENT_CSO,
    uiFrequency := 250,
    uiDitherFrequency := 125,
    uiDitherValue := 0,
    usiKP := 50,
    usiKI := 50,
    uiStartRatio := 500,
    StateData := NVL_UDP_RX.All.OUT0002,
    Output_Enable := ENABLE_OUTPUTS_COMMON,
    GRP_OUTPUT_DIAG := NVL_UDP_TX.All_Outputs_Diag.GROUP0,
    IO_CRXXXX_OUTPUT_DIAG := NVL_UDP_TX.All_Outputs_Diag.OUT0002); // CRXXXX_OUTPUT_PWM_FB

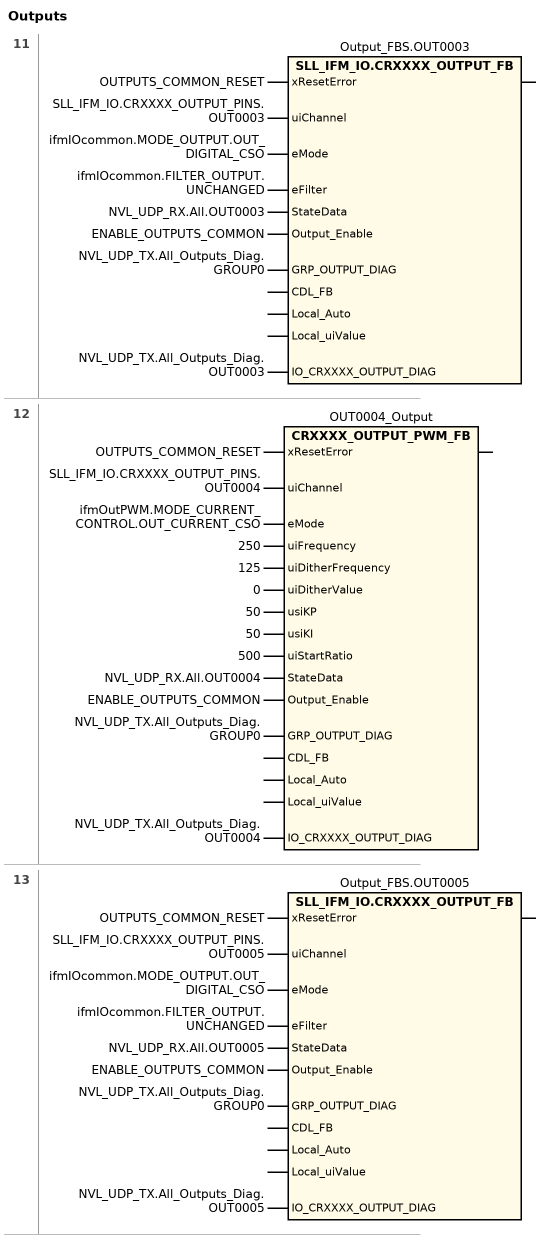
// NETWORK 11
Output_FBS.OUT0003(
    xResetError := OUTPUTS_COMMON_RESET,
    uiChannel := SLL_IFM_IO.CRXXXX_OUTPUT_PINS.OUT0003,
    eMode := ifmIOcommon.MODE_OUTPUT.OUT_DIGITAL_CSO,
    eFilter := ifmIOcommon.FILTER_OUTPUT.UNCHANGED,
    StateData := NVL_UDP_RX.All.OUT0003,
    Output_Enable := ENABLE_OUTPUTS_COMMON,
    GRP_OUTPUT_DIAG := NVL_UDP_TX.All_Outputs_Diag.GROUP0,
    IO_CRXXXX_OUTPUT_DIAG := NVL_UDP_TX.All_Outputs_Diag.OUT0003); // SLL_IFM_IO.CRXXXX_OUTPUT_FB

// NETWORK 12
OUT0004_Output(
    xResetError := OUTPUTS_COMMON_RESET,
    uiChannel := SLL_IFM_IO.CRXXXX_OUTPUT_PINS.OUT0004,
    eMode := ifmOutPWM.MODE_CURRENT_CONTROL.OUT_CURRENT_CSO,
    uiFrequency := 250,
    uiDitherFrequency := 125,
    uiDitherValue := 0,
    usiKP := 50,
    usiKI := 50,
    uiStartRatio := 500,
    StateData := NVL_UDP_RX.All.OUT0004,
    Output_Enable := ENABLE_OUTPUTS_COMMON,
    GRP_OUTPUT_DIAG := NVL_UDP_TX.All_Outputs_Diag.GROUP0,
    IO_CRXXXX_OUTPUT_DIAG := NVL_UDP_TX.All_Outputs_Diag.OUT0004); // CRXXXX_OUTPUT_PWM_FB

// NETWORK 13
Output_FBS.OUT0005(
    xResetError := OUTPUTS_COMMON_RESET,
    uiChannel := SLL_IFM_IO.CRXXXX_OUTPUT_PINS.OUT0005,
    eMode := ifmIOcommon.MODE_OUTPUT.OUT_DIGITAL_CSO,
    eFilter := ifmIOcommon.FILTER_OUTPUT.UNCHANGED,
    StateData := NVL_UDP_RX.All.OUT0005,
    Output_Enable := ENABLE_OUTPUTS_COMMON,
    GRP_OUTPUT_DIAG := NVL_UDP_TX.All_Outputs_Diag.GROUP0,
    IO_CRXXXX_OUTPUT_DIAG := NVL_UDP_TX.All_Outputs_Diag.OUT0005); // SLL_IFM_IO.CRXXXX_OUTPUT_FB

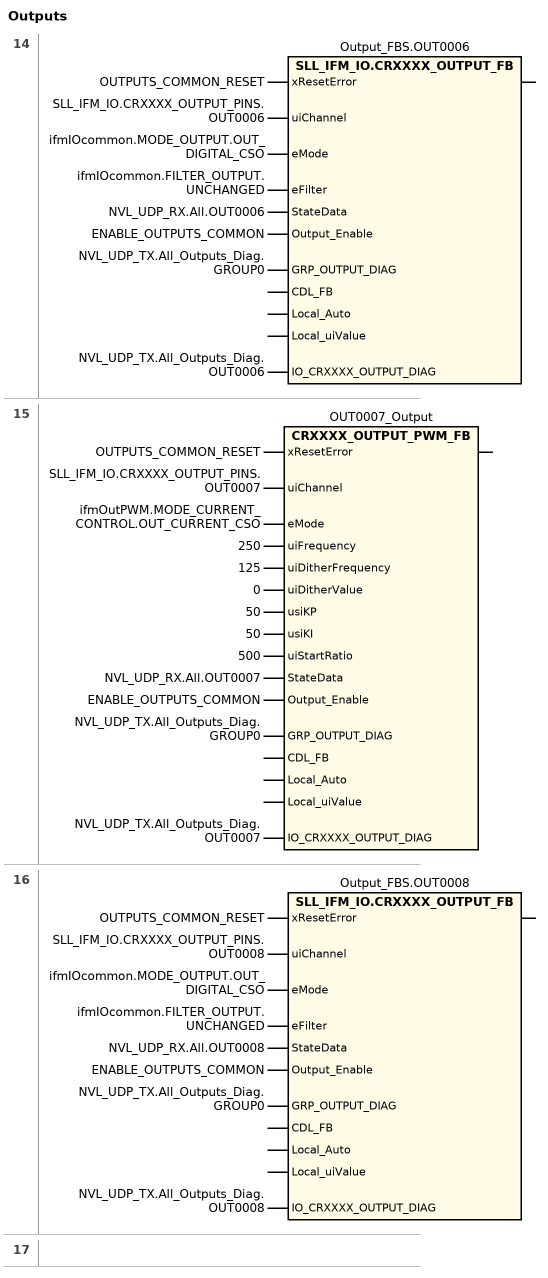
// NETWORK 14
Output_FBS.OUT0006(
    xResetError := OUTPUTS_COMMON_RESET,
    uiChannel := SLL_IFM_IO.CRXXXX_OUTPUT_PINS.OUT0006,
    eMode := ifmIOcommon.MODE_OUTPUT.OUT_DIGITAL_CSO,
    eFilter := ifmIOcommon.FILTER_OUTPUT.UNCHANGED,
    StateData := NVL_UDP_RX.All.OUT0006,
    Output_Enable := ENABLE_OUTPUTS_COMMON,
    GRP_OUTPUT_DIAG := NVL_UDP_TX.All_Outputs_Diag.GROUP0,
    IO_CRXXXX_OUTPUT_DIAG := NVL_UDP_TX.All_Outputs_Diag.OUT0006); // SLL_IFM_IO.CRXXXX_OUTPUT_FB

// NETWORK 15
OUT0007_Output(
    xResetError := OUTPUTS_COMMON_RESET,
    uiChannel := SLL_IFM_IO.CRXXXX_OUTPUT_PINS.OUT0007,
    eMode := ifmOutPWM.MODE_CURRENT_CONTROL.OUT_CURRENT_CSO,
    uiFrequency := 250,
    uiDitherFrequency := 125,
    uiDitherValue := 0,
    usiKP := 50,
    usiKI := 50,
    uiStartRatio := 500,
    StateData := NVL_UDP_RX.All.OUT0007,
    Output_Enable := ENABLE_OUTPUTS_COMMON,
    GRP_OUTPUT_DIAG := NVL_UDP_TX.All_Outputs_Diag.GROUP0,
    IO_CRXXXX_OUTPUT_DIAG := NVL_UDP_TX.All_Outputs_Diag.OUT0007); // CRXXXX_OUTPUT_PWM_FB

// NETWORK 16
Output_FBS.OUT0008(
    xResetError := OUTPUTS_COMMON_RESET,
    uiChannel := SLL_IFM_IO.CRXXXX_OUTPUT_PINS.OUT0008,
    eMode := ifmIOcommon.MODE_OUTPUT.OUT_DIGITAL_CSO,
    eFilter := ifmIOcommon.FILTER_OUTPUT.UNCHANGED,
    StateData := NVL_UDP_RX.All.OUT0008,
    Output_Enable := ENABLE_OUTPUTS_COMMON,
    GRP_OUTPUT_DIAG := NVL_UDP_TX.All_Outputs_Diag.GROUP0,
    IO_CRXXXX_OUTPUT_DIAG := NVL_UDP_TX.All_Outputs_Diag.OUT0008); // SLL_IFM_IO.CRXXXX_OUTPUT_FB

// NETWORK 17

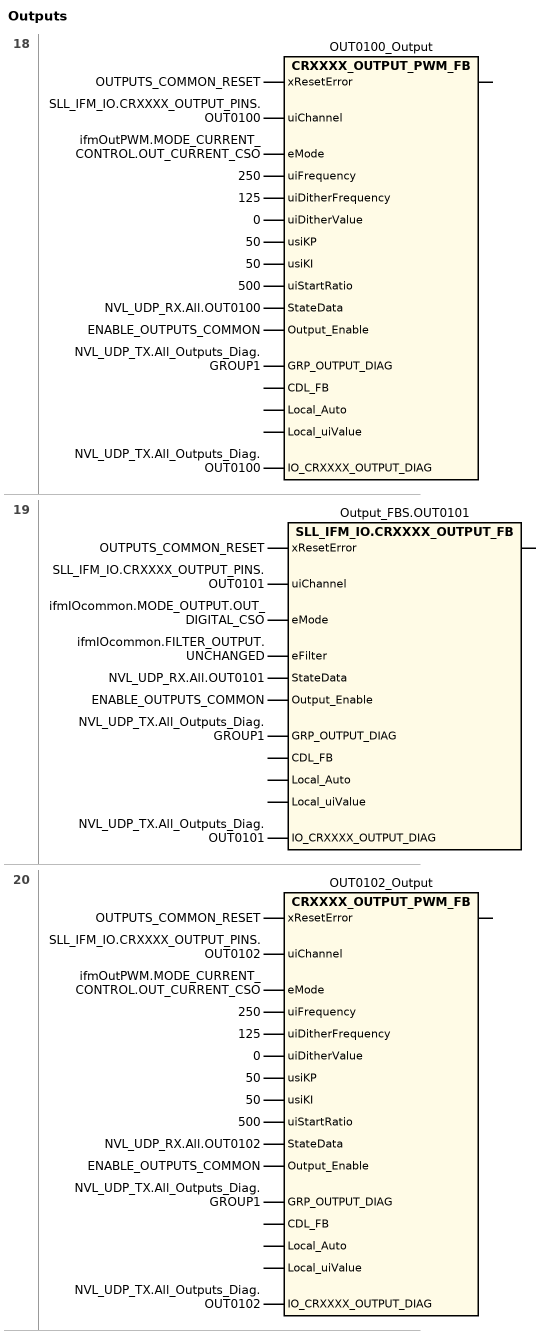
// NETWORK 18
OUT0100_Output(
    xResetError := OUTPUTS_COMMON_RESET,
    uiChannel := SLL_IFM_IO.CRXXXX_OUTPUT_PINS.OUT0100,
    eMode := ifmOutPWM.MODE_CURRENT_CONTROL.OUT_CURRENT_CSO,
    uiFrequency := 250,
    uiDitherFrequency := 125,
    uiDitherValue := 0,
    usiKP := 50,
    usiKI := 50,
    uiStartRatio := 500,
    StateData := NVL_UDP_RX.All.OUT0100,
    Output_Enable := ENABLE_OUTPUTS_COMMON,
    GRP_OUTPUT_DIAG := NVL_UDP_TX.All_Outputs_Diag.GROUP1,
    IO_CRXXXX_OUTPUT_DIAG := NVL_UDP_TX.All_Outputs_Diag.OUT0100); // CRXXXX_OUTPUT_PWM_FB

// NETWORK 19
Output_FBS.OUT0101(
    xResetError := OUTPUTS_COMMON_RESET,
    uiChannel := SLL_IFM_IO.CRXXXX_OUTPUT_PINS.OUT0101,
    eMode := ifmIOcommon.MODE_OUTPUT.OUT_DIGITAL_CSO,
    eFilter := ifmIOcommon.FILTER_OUTPUT.UNCHANGED,
    StateData := NVL_UDP_RX.All.OUT0101,
    Output_Enable := ENABLE_OUTPUTS_COMMON,
    GRP_OUTPUT_DIAG := NVL_UDP_TX.All_Outputs_Diag.GROUP1,
    IO_CRXXXX_OUTPUT_DIAG := NVL_UDP_TX.All_Outputs_Diag.OUT0101); // SLL_IFM_IO.CRXXXX_OUTPUT_FB

// NETWORK 20
OUT0102_Output(
    xResetError := OUTPUTS_COMMON_RESET,
    uiChannel := SLL_IFM_IO.CRXXXX_OUTPUT_PINS.OUT0102,
    eMode := ifmOutPWM.MODE_CURRENT_CONTROL.OUT_CURRENT_CSO,
    uiFrequency := 250,
    uiDitherFrequency := 125,
    uiDitherValue := 0,
    usiKP := 50,
    usiKI := 50,
    uiStartRatio := 500,
    StateData := NVL_UDP_RX.All.OUT0102,
    Output_Enable := ENABLE_OUTPUTS_COMMON,
    GRP_OUTPUT_DIAG := NVL_UDP_TX.All_Outputs_Diag.GROUP1,
    IO_CRXXXX_OUTPUT_DIAG := NVL_UDP_TX.All_Outputs_Diag.OUT0102); // CRXXXX_OUTPUT_PWM_FB

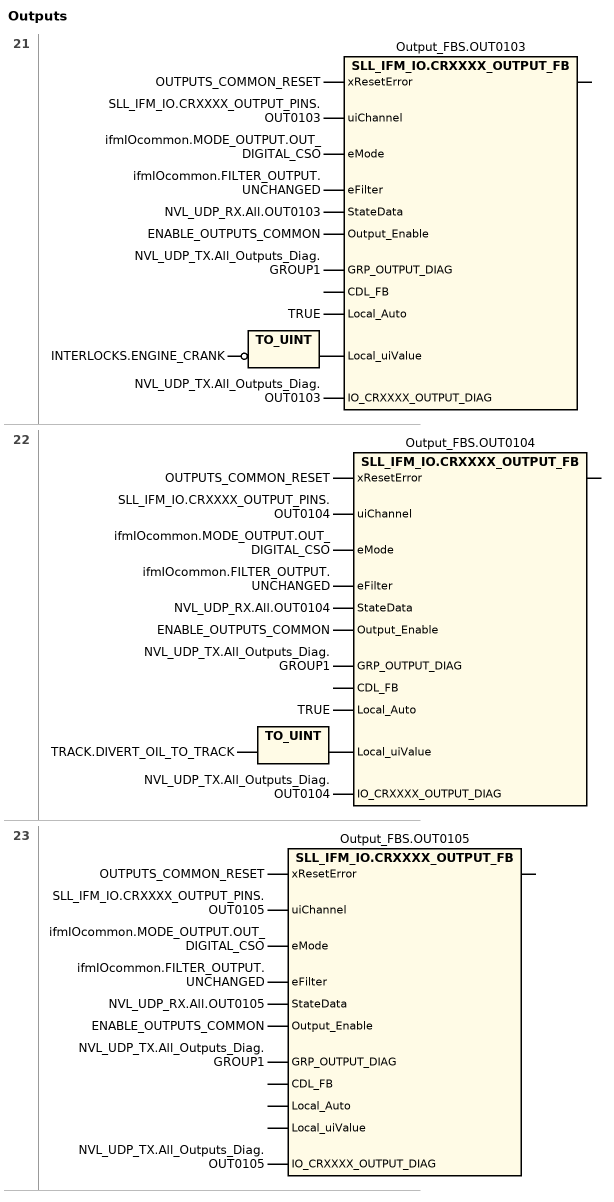
// NETWORK 21
Output_FBS.OUT0103(
    xResetError := OUTPUTS_COMMON_RESET,
    uiChannel := SLL_IFM_IO.CRXXXX_OUTPUT_PINS.OUT0103,
    eMode := ifmIOcommon.MODE_OUTPUT.OUT_DIGITAL_CSO,
    eFilter := ifmIOcommon.FILTER_OUTPUT.UNCHANGED,
    StateData := NVL_UDP_RX.All.OUT0103,
    Output_Enable := ENABLE_OUTPUTS_COMMON,
    GRP_OUTPUT_DIAG := NVL_UDP_TX.All_Outputs_Diag.GROUP1,
    Local_Auto := TRUE,
    Local_uiValue := TO_UINT(NOT INTERLOCKS.ENGINE_CRANK),
    IO_CRXXXX_OUTPUT_DIAG := NVL_UDP_TX.All_Outputs_Diag.OUT0103); // SLL_IFM_IO.CRXXXX_OUTPUT_FB

// NETWORK 22
Output_FBS.OUT0104(
    xResetError := OUTPUTS_COMMON_RESET,
    uiChannel := SLL_IFM_IO.CRXXXX_OUTPUT_PINS.OUT0104,
    eMode := ifmIOcommon.MODE_OUTPUT.OUT_DIGITAL_CSO,
    eFilter := ifmIOcommon.FILTER_OUTPUT.UNCHANGED,
    StateData := NVL_UDP_RX.All.OUT0104,
    Output_Enable := ENABLE_OUTPUTS_COMMON,
    GRP_OUTPUT_DIAG := NVL_UDP_TX.All_Outputs_Diag.GROUP1,
    Local_Auto := TRUE,
    Local_uiValue := TO_UINT(TRACK.DIVERT_OIL_TO_TRACK),
    IO_CRXXXX_OUTPUT_DIAG := NVL_UDP_TX.All_Outputs_Diag.OUT0104); // SLL_IFM_IO.CRXXXX_OUTPUT_FB

// NETWORK 23
Output_FBS.OUT0105(
    xResetError := OUTPUTS_COMMON_RESET,
    uiChannel := SLL_IFM_IO.CRXXXX_OUTPUT_PINS.OUT0105,
    eMode := ifmIOcommon.MODE_OUTPUT.OUT_DIGITAL_CSO,
    eFilter := ifmIOcommon.FILTER_OUTPUT.UNCHANGED,
    StateData := NVL_UDP_RX.All.OUT0105,
    Output_Enable := ENABLE_OUTPUTS_COMMON,
    GRP_OUTPUT_DIAG := NVL_UDP_TX.All_Outputs_Diag.GROUP1,
    IO_CRXXXX_OUTPUT_DIAG := NVL_UDP_TX.All_Outputs_Diag.OUT0105); // SLL_IFM_IO.CRXXXX_OUTPUT_FB

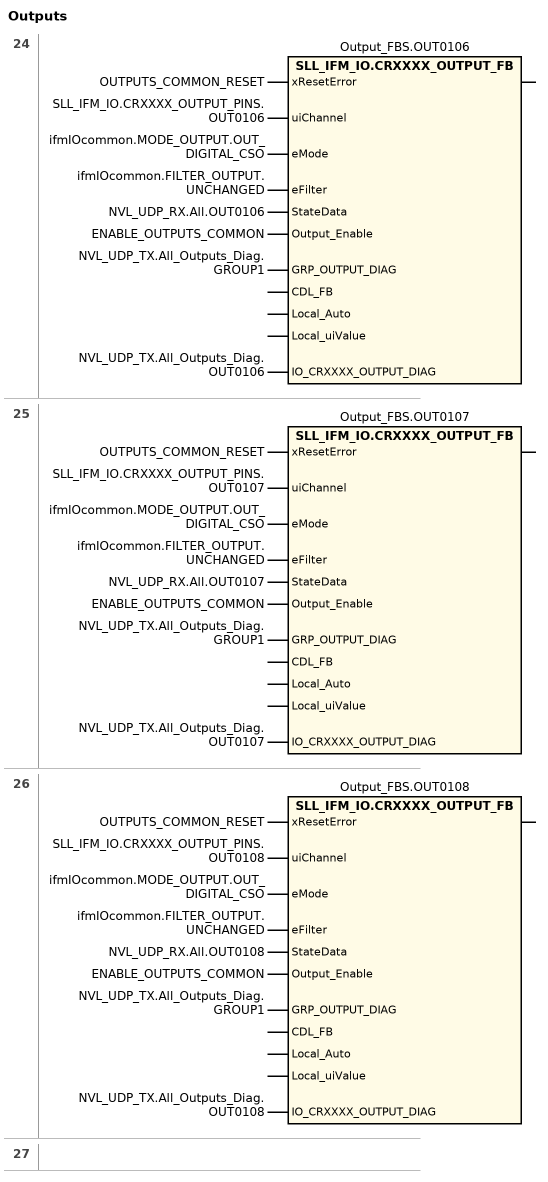
// NETWORK 24
Output_FBS.OUT0106(
    xResetError := OUTPUTS_COMMON_RESET,
    uiChannel := SLL_IFM_IO.CRXXXX_OUTPUT_PINS.OUT0106,
    eMode := ifmIOcommon.MODE_OUTPUT.OUT_DIGITAL_CSO,
    eFilter := ifmIOcommon.FILTER_OUTPUT.UNCHANGED,
    StateData := NVL_UDP_RX.All.OUT0106,
    Output_Enable := ENABLE_OUTPUTS_COMMON,
    GRP_OUTPUT_DIAG := NVL_UDP_TX.All_Outputs_Diag.GROUP1,
    IO_CRXXXX_OUTPUT_DIAG := NVL_UDP_TX.All_Outputs_Diag.OUT0106); // SLL_IFM_IO.CRXXXX_OUTPUT_FB

// NETWORK 25
Output_FBS.OUT0107(
    xResetError := OUTPUTS_COMMON_RESET,
    uiChannel := SLL_IFM_IO.CRXXXX_OUTPUT_PINS.OUT0107,
    eMode := ifmIOcommon.MODE_OUTPUT.OUT_DIGITAL_CSO,
    eFilter := ifmIOcommon.FILTER_OUTPUT.UNCHANGED,
    StateData := NVL_UDP_RX.All.OUT0107,
    Output_Enable := ENABLE_OUTPUTS_COMMON,
    GRP_OUTPUT_DIAG := NVL_UDP_TX.All_Outputs_Diag.GROUP1,
    IO_CRXXXX_OUTPUT_DIAG := NVL_UDP_TX.All_Outputs_Diag.OUT0107); // SLL_IFM_IO.CRXXXX_OUTPUT_FB

// NETWORK 26
Output_FBS.OUT0108(
    xResetError := OUTPUTS_COMMON_RESET,
    uiChannel := SLL_IFM_IO.CRXXXX_OUTPUT_PINS.OUT0108,
    eMode := ifmIOcommon.MODE_OUTPUT.OUT_DIGITAL_CSO,
    eFilter := ifmIOcommon.FILTER_OUTPUT.UNCHANGED,
    StateData := NVL_UDP_RX.All.OUT0108,
    Output_Enable := ENABLE_OUTPUTS_COMMON,
    GRP_OUTPUT_DIAG := NVL_UDP_TX.All_Outputs_Diag.GROUP1,
    IO_CRXXXX_OUTPUT_DIAG := NVL_UDP_TX.All_Outputs_Diag.OUT0108); // SLL_IFM_IO.CRXXXX_OUTPUT_FB

// NETWORK 27

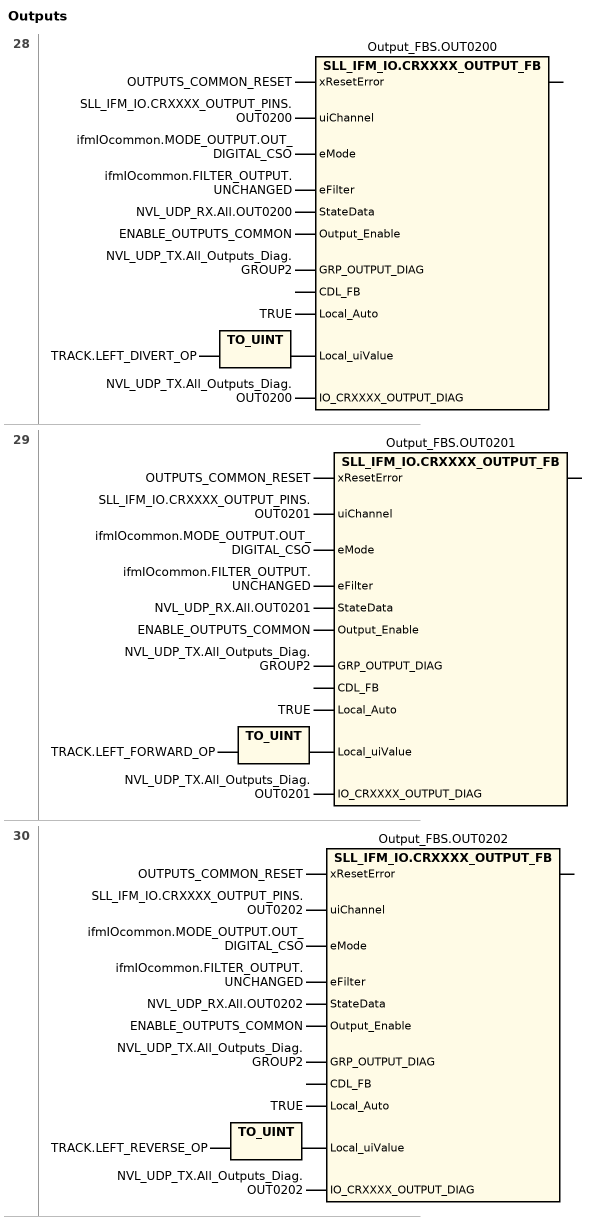
// NETWORK 28
Output_FBS.OUT0200(
    xResetError := OUTPUTS_COMMON_RESET,
    uiChannel := SLL_IFM_IO.CRXXXX_OUTPUT_PINS.OUT0200,
    eMode := ifmIOcommon.MODE_OUTPUT.OUT_DIGITAL_CSO,
    eFilter := ifmIOcommon.FILTER_OUTPUT.UNCHANGED,
    StateData := NVL_UDP_RX.All.OUT0200,
    Output_Enable := ENABLE_OUTPUTS_COMMON,
    GRP_OUTPUT_DIAG := NVL_UDP_TX.All_Outputs_Diag.GROUP2,
    Local_Auto := TRUE,
    Local_uiValue := TO_UINT(TRACK.LEFT_DIVERT_OP),
    IO_CRXXXX_OUTPUT_DIAG := NVL_UDP_TX.All_Outputs_Diag.OUT0200); // SLL_IFM_IO.CRXXXX_OUTPUT_FB

// NETWORK 29
Output_FBS.OUT0201(
    xResetError := OUTPUTS_COMMON_RESET,
    uiChannel := SLL_IFM_IO.CRXXXX_OUTPUT_PINS.OUT0201,
    eMode := ifmIOcommon.MODE_OUTPUT.OUT_DIGITAL_CSO,
    eFilter := ifmIOcommon.FILTER_OUTPUT.UNCHANGED,
    StateData := NVL_UDP_RX.All.OUT0201,
    Output_Enable := ENABLE_OUTPUTS_COMMON,
    GRP_OUTPUT_DIAG := NVL_UDP_TX.All_Outputs_Diag.GROUP2,
    Local_Auto := TRUE,
    Local_uiValue := TO_UINT(TRACK.LEFT_FORWARD_OP),
    IO_CRXXXX_OUTPUT_DIAG := NVL_UDP_TX.All_Outputs_Diag.OUT0201); // SLL_IFM_IO.CRXXXX_OUTPUT_FB

// NETWORK 30
Output_FBS.OUT0202(
    xResetError := OUTPUTS_COMMON_RESET,
    uiChannel := SLL_IFM_IO.CRXXXX_OUTPUT_PINS.OUT0202,
    eMode := ifmIOcommon.MODE_OUTPUT.OUT_DIGITAL_CSO,
    eFilter := ifmIOcommon.FILTER_OUTPUT.UNCHANGED,
    StateData := NVL_UDP_RX.All.OUT0202,
    Output_Enable := ENABLE_OUTPUTS_COMMON,
    GRP_OUTPUT_DIAG := NVL_UDP_TX.All_Outputs_Diag.GROUP2,
    Local_Auto := TRUE,
    Local_uiValue := TO_UINT(TRACK.LEFT_REVERSE_OP),
    IO_CRXXXX_OUTPUT_DIAG := NVL_UDP_TX.All_Outputs_Diag.OUT0202); // SLL_IFM_IO.CRXXXX_OUTPUT_FB

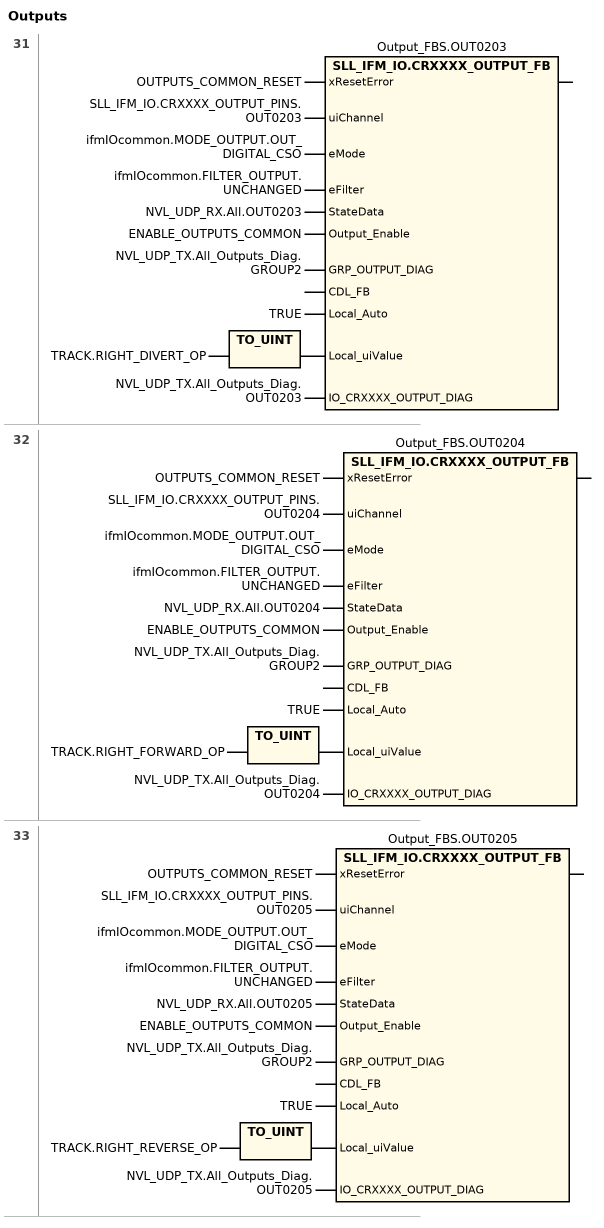
// NETWORK 31
Output_FBS.OUT0203(
    xResetError := OUTPUTS_COMMON_RESET,
    uiChannel := SLL_IFM_IO.CRXXXX_OUTPUT_PINS.OUT0203,
    eMode := ifmIOcommon.MODE_OUTPUT.OUT_DIGITAL_CSO,
    eFilter := ifmIOcommon.FILTER_OUTPUT.UNCHANGED,
    StateData := NVL_UDP_RX.All.OUT0203,
    Output_Enable := ENABLE_OUTPUTS_COMMON,
    GRP_OUTPUT_DIAG := NVL_UDP_TX.All_Outputs_Diag.GROUP2,
    Local_Auto := TRUE,
    Local_uiValue := TO_UINT(TRACK.RIGHT_DIVERT_OP),
    IO_CRXXXX_OUTPUT_DIAG := NVL_UDP_TX.All_Outputs_Diag.OUT0203); // SLL_IFM_IO.CRXXXX_OUTPUT_FB

// NETWORK 32
Output_FBS.OUT0204(
    xResetError := OUTPUTS_COMMON_RESET,
    uiChannel := SLL_IFM_IO.CRXXXX_OUTPUT_PINS.OUT0204,
    eMode := ifmIOcommon.MODE_OUTPUT.OUT_DIGITAL_CSO,
    eFilter := ifmIOcommon.FILTER_OUTPUT.UNCHANGED,
    StateData := NVL_UDP_RX.All.OUT0204,
    Output_Enable := ENABLE_OUTPUTS_COMMON,
    GRP_OUTPUT_DIAG := NVL_UDP_TX.All_Outputs_Diag.GROUP2,
    Local_Auto := TRUE,
    Local_uiValue := TO_UINT(TRACK.RIGHT_FORWARD_OP),
    IO_CRXXXX_OUTPUT_DIAG := NVL_UDP_TX.All_Outputs_Diag.OUT0204); // SLL_IFM_IO.CRXXXX_OUTPUT_FB

// NETWORK 33
Output_FBS.OUT0205(
    xResetError := OUTPUTS_COMMON_RESET,
    uiChannel := SLL_IFM_IO.CRXXXX_OUTPUT_PINS.OUT0205,
    eMode := ifmIOcommon.MODE_OUTPUT.OUT_DIGITAL_CSO,
    eFilter := ifmIOcommon.FILTER_OUTPUT.UNCHANGED,
    StateData := NVL_UDP_RX.All.OUT0205,
    Output_Enable := ENABLE_OUTPUTS_COMMON,
    GRP_OUTPUT_DIAG := NVL_UDP_TX.All_Outputs_Diag.GROUP2,
    Local_Auto := TRUE,
    Local_uiValue := TO_UINT(TRACK.RIGHT_REVERSE_OP),
    IO_CRXXXX_OUTPUT_DIAG := NVL_UDP_TX.All_Outputs_Diag.OUT0205); // SLL_IFM_IO.CRXXXX_OUTPUT_FB

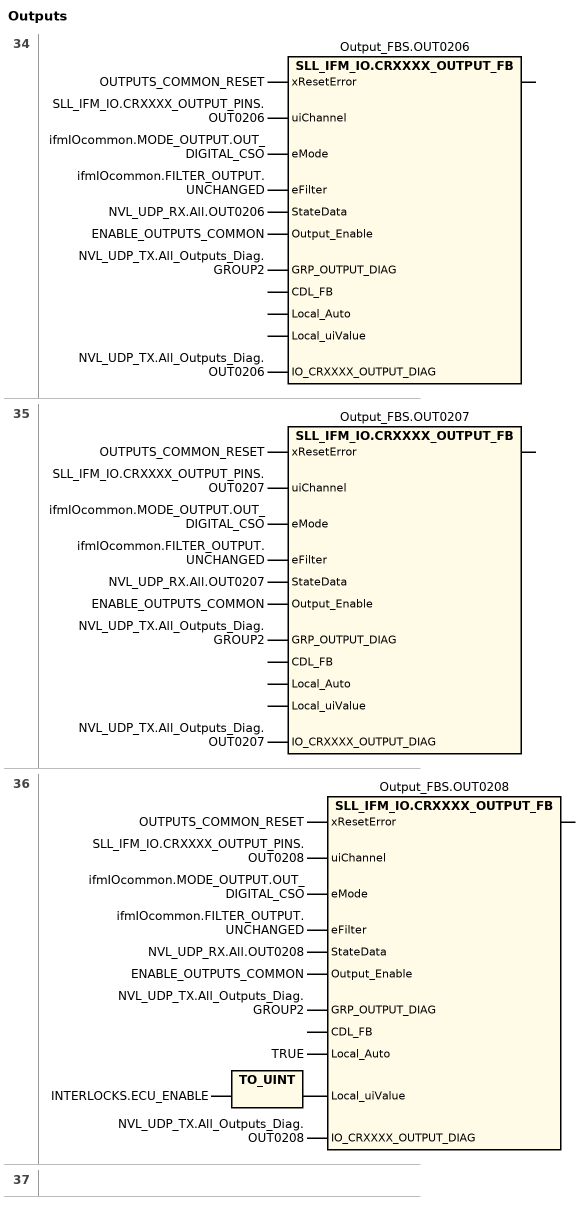
// NETWORK 34
Output_FBS.OUT0206(
    xResetError := OUTPUTS_COMMON_RESET,
    uiChannel := SLL_IFM_IO.CRXXXX_OUTPUT_PINS.OUT0206,
    eMode := ifmIOcommon.MODE_OUTPUT.OUT_DIGITAL_CSO,
    eFilter := ifmIOcommon.FILTER_OUTPUT.UNCHANGED,
    StateData := NVL_UDP_RX.All.OUT0206,
    Output_Enable := ENABLE_OUTPUTS_COMMON,
    GRP_OUTPUT_DIAG := NVL_UDP_TX.All_Outputs_Diag.GROUP2,
    IO_CRXXXX_OUTPUT_DIAG := NVL_UDP_TX.All_Outputs_Diag.OUT0206); // SLL_IFM_IO.CRXXXX_OUTPUT_FB

// NETWORK 35
Output_FBS.OUT0207(
    xResetError := OUTPUTS_COMMON_RESET,
    uiChannel := SLL_IFM_IO.CRXXXX_OUTPUT_PINS.OUT0207,
    eMode := ifmIOcommon.MODE_OUTPUT.OUT_DIGITAL_CSO,
    eFilter := ifmIOcommon.FILTER_OUTPUT.UNCHANGED,
    StateData := NVL_UDP_RX.All.OUT0207,
    Output_Enable := ENABLE_OUTPUTS_COMMON,
    GRP_OUTPUT_DIAG := NVL_UDP_TX.All_Outputs_Diag.GROUP2,
    IO_CRXXXX_OUTPUT_DIAG := NVL_UDP_TX.All_Outputs_Diag.OUT0207); // SLL_IFM_IO.CRXXXX_OUTPUT_FB

// NETWORK 36
Output_FBS.OUT0208(
    xResetError := OUTPUTS_COMMON_RESET,
    uiChannel := SLL_IFM_IO.CRXXXX_OUTPUT_PINS.OUT0208,
    eMode := ifmIOcommon.MODE_OUTPUT.OUT_DIGITAL_CSO,
    eFilter := ifmIOcommon.FILTER_OUTPUT.UNCHANGED,
    StateData := NVL_UDP_RX.All.OUT0208,
    Output_Enable := ENABLE_OUTPUTS_COMMON,
    GRP_OUTPUT_DIAG := NVL_UDP_TX.All_Outputs_Diag.GROUP2,
    Local_Auto := TRUE,
    Local_uiValue := TO_UINT(INTERLOCKS.ECU_ENABLE),
    IO_CRXXXX_OUTPUT_DIAG := NVL_UDP_TX.All_Outputs_Diag.OUT0208); // SLL_IFM_IO.CRXXXX_OUTPUT_FB

// NETWORK 37

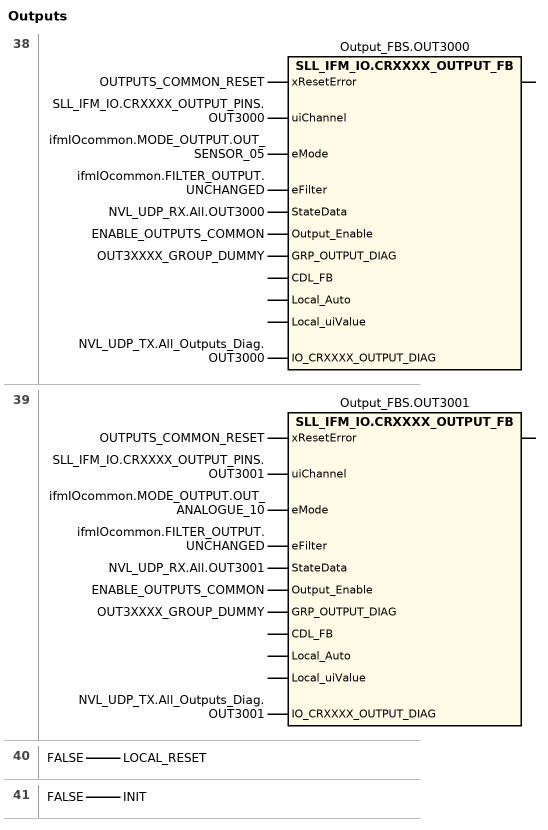
// NETWORK 38
Output_FBS.OUT3000(
    xResetError := OUTPUTS_COMMON_RESET,
    uiChannel := SLL_IFM_IO.CRXXXX_OUTPUT_PINS.OUT3000,
    eMode := ifmIOcommon.MODE_OUTPUT.OUT_SENSOR_05,
    eFilter := ifmIOcommon.FILTER_OUTPUT.UNCHANGED,
    StateData := NVL_UDP_RX.All.OUT3000,
    Output_Enable := ENABLE_OUTPUTS_COMMON,
    GRP_OUTPUT_DIAG := OUT3XXXX_GROUP_DUMMY,
    IO_CRXXXX_OUTPUT_DIAG := NVL_UDP_TX.All_Outputs_Diag.OUT3000); // SLL_IFM_IO.CRXXXX_OUTPUT_FB

// NETWORK 39
Output_FBS.OUT3001(
    xResetError := OUTPUTS_COMMON_RESET,
    uiChannel := SLL_IFM_IO.CRXXXX_OUTPUT_PINS.OUT3001,
    eMode := ifmIOcommon.MODE_OUTPUT.OUT_ANALOGUE_10,
    eFilter := ifmIOcommon.FILTER_OUTPUT.UNCHANGED,
    StateData := NVL_UDP_RX.All.OUT3001,
    Output_Enable := ENABLE_OUTPUTS_COMMON,
    GRP_OUTPUT_DIAG := OUT3XXXX_GROUP_DUMMY,
    IO_CRXXXX_OUTPUT_DIAG := NVL_UDP_TX.All_Outputs_Diag.OUT3001); // SLL_IFM_IO.CRXXXX_OUTPUT_FB

// NETWORK 40
LOCAL_RESET := FALSE;

// NETWORK 41
INIT := FALSE;

END_PROGRAM

// StandardPLC/Application/Outputs/CRXXXX_OUTPUT_PWM_FB
FUNCTION_BLOCK CRXXXX_OUTPUT_PWM_FB
VAR_INPUT
	xResetError:BOOL;
	uiChannel:WORD;	
	eMode: ifmOutPWM.MODE_CURRENT_CONTROL;
	uiFrequency: UINT; 
	uiDitherFrequency: UINT;	 
	uiDitherValue: UINT;	 
	usiKP: USINT;	 
	usiKI: USINT;	 
	uiStartRatio: UINT;	
	StateData: CRXXXX_OUTPUT_STATE_DATA;
	Output_Enable: BOOL;
	GRP_OUTPUT_DIAG: REFERENCE TO CRXXXX_OUTPUT_GROUP_DATA;
	CDL_FB: ifmIOconfigDiagProt.ConfigDiagLevel;
	Local_Auto: BOOL:=FALSE;
	Local_uiValue: UINT:=0;	
END_VAR
VAR_OUTPUT
END_VAR
VAR
	Output_FB: ifmOutPWM.CurrentControl;	
END_VAR

VAR_IN_OUT
	IO_CRXXXX_OUTPUT_DIAG: CRXXXX_OUTPUT_DATA;
END_VAR

